# B&R Automation Studio project DeltaTestowa1
Automation Studio 4.12.6.106; technology packages: mapp 5.24.2, mappMotion 5.26.1, mappView 5.24.2

## Configuration Config1

CPU 5APC3100.KBU0-000, AutomationRuntime J4.93, Build 4.1.2, Safety 0.0, Vc V4.73.2

CPU 5APC3100.KBU1-000, AutomationRuntime J4.93, Build 4.1.2, Safety 0.0, Vc V4.73.2

CPU 5APC3100.KBU2-000, AutomationRuntime C4.90, Build 4.1.2, Safety 0.0, Vc 

CPU X20CP1584, AutomationRuntime J4.93, Build 4.1.2, Vc V4.73.2

### Task classes (Cpu.sw)
```
Cyclic#4:
  Program <- Program.prg
Libraries: McBase, MpBase, MpRobotics, McAxGroup, McPathGen, McAxis, McProgInt, McAcpAx, McPureVAx
```

### Task classes (Cpu.sw)
```
Cyclic#1:
  PrgPick <- PickAndPlace.PrgPick.prg
  PrgPickCor <- PickAndPlace.PrgPickCore.prg
  PrgMechs <- PickAndPlace.PrgMechs.prg
  PrgPlace <- PickAndPlace.PrgPlace.prg
Cyclic#4:
  Program <- Program.prg
DataObjects: McAcpSys
NcDataObjects: McDriveLog
Binaries: McAcpDrv, udbdef, McAcpSim, mvLoader, arflatprv, TCData, McProfGen, mCoWebSc, McMechSys, FWRules, arcoal, arsvcreg, Settings, iomap, Config_3, Config_4, Role, ashwac, Config_10, asfw, Config_5, sysconf, Config_2, arconfig, Config_6, Config_8, Config_1, Hierarchy, ashwd, Config_7, User, Config_9
Libraries: UserLib, McBase, MpBase, MpRobotics, McAxGroup, McPathGen, McAxis, McProgInt, McAcpAx, CoTrace, AsZip, FileIO, runtime, MpAxis, asarprof, asieccon, asarlog, asio, asmem, astime, asepl, dataobj, brsystem, arssl, sys_lib, powerlnk, mctrkpath, mppick, MpAlarm
```

### Task classes (Cpu.sw)
```
Cyclic#1:
  PrgPickCor <- PickAndPlace.PrgPickCore.prg
Cyclic#2:
  PrgPick <- PickAndPlace.PrgPick.prg
  PrgPlace <- PickAndPlace.PrgPlace.prg
Cyclic#3:
  PrgMechs <- PickAndPlace.PrgMechs.prg
DataObjects: McAcpSys
NcDataObjects: McDriveLog
Binaries: McAcpDrv, udbdef, McAcpSim, mvLoader, arflatprv, TCData, McProfGen, mCoWebSc, McMechSys, FWRules, arcoal, arsvcreg, OpcUaSrv, Settings, iomap, Config_3, Config_4, Role, ashwac, Config_10, asfw, Config_5, sysconf, Config_2, arconfig, Config_6, Config_8, Config_1, Hierarchy, ashwd, Config_7, User, Config_9
Libraries: UserLib, McBase, MpBase, MpRobotics, McAxGroup, McPathGen, McAxis, McProgInt, McAcpAx, CoTrace, AsZip, FileIO, runtime, MpAxis, McAcpPar, McTrkPath, MpPick, McAcpTrak, MpCnc, MpTool, sys_lib, McDS402Ax, McPureVAx, McStpAx, MpServer, AsIODiag, asarprof, asarlog, asio, asmem, astime, asepl, dataobj, brsystem, arssl, powerlnk, asioacc, aruser, asieccon
```

### Task classes (Cpu1.sw)
```

```

### Task classes (Cpu.sw)
```
Cyclic#4:
  Program <- Program.prg
Libraries: McBase, MpBase, MpRobotics, McAxGroup, McPathGen, McAxis, McProgInt, McAcpAx
```

### Hardware
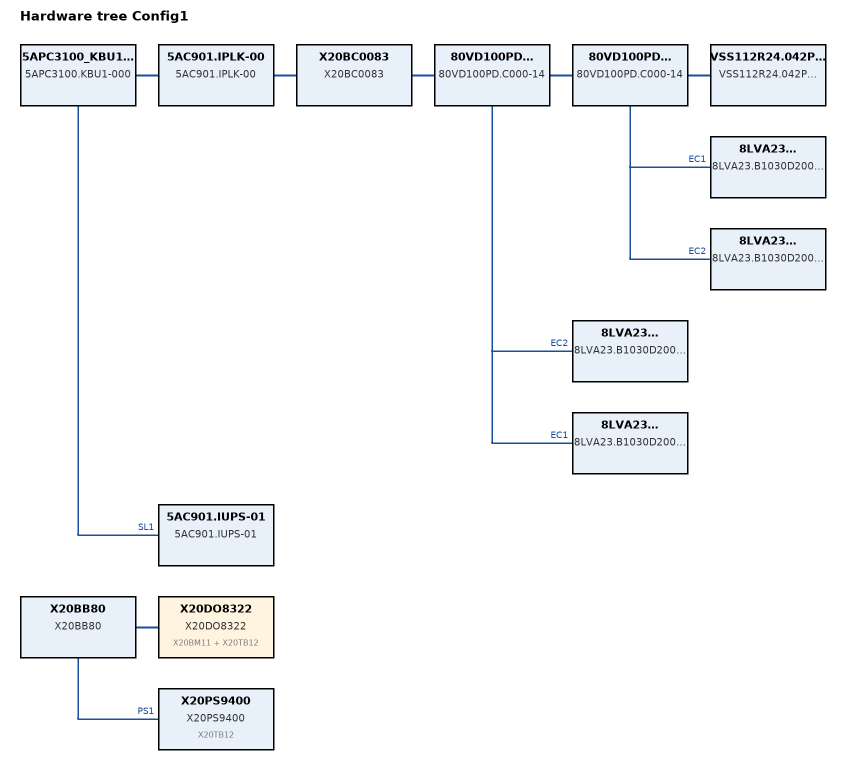
```
5AC901.IPLK-00 : 5AC901.IPLK-00 v1.8.0.1  [SL -> 5APC3100_KBU1_000a.SL2]
  Connector IF1:
    MtuSize = 1500
    CycleTime = 400
    Channel1
    ChannelID1 = McAcpBroadcast
    ChannelType1 = OCTET[36]
    InternetAddress = 192.168.200.240
    SubnetMask = 255.255.255.0
5AC901.IUPS-01 : 5AC901.IUPS-01 v1.3.1.0  [SL -> 5APC3100_KBU1_000a.SL1]
5APC3100_KBU1_000a : 5APC3100.KBU1-000 v2.2.1.0
  Connector IF3:
    AssignedOperatingSystem = ARemb
    ActivateDevice = 1
    Mode = Manual
    InternetAddress = 192.168.0.20
    SubnetMask = 255.255.255.0
    ActivateSnmp = 2
  Connector IF4:
    AssignedOperatingSystem = ARemb
    ActivateDevice = 1
    Mode = Manual
    InternetAddress = 10.0.0.20
    SubnetMask = 255.255.255.0
    ActivateSnmp = 2
  Connector IF5:
    AssignedOperatingSystem = ARemb
  Connector IF6:
    AssignedOperatingSystem = ARemb
  Connector IF7:
    AssignedOperatingSystem = ARemb
  Connector IF8:
    AssignedOperatingSystem = ARemb
  ConfigurationID = Proj_Config1
  MotionLoggerSize = 2048000
  TimerDeviceType = EPLX2X
  TimerDevice = 5AC901.IPLK-00.IF1
  TaskClassIdleTime = 2000
  Cyclic1Tolerance = 0
  FileDevice1
  FileDeviceName1 = CNC_PrgDir
  FileDevicePath1 = C:\CNC_PrgDir\
  FileDevice2
  FileDeviceName2 = CF
  FileDevicePath2 = C:\CF\
  FileDevice3
  FileDeviceName3 = CNC_PrgDirRobot
  FileDevicePath3 = F:\CNC_PrgDirRobot
  ActivateOpcUa = 1
  OpcUaPort = 4841
  OpcUaInformationModels_PV_Version = 1
80VD100PD.C000-14 : 80VD100PD.C000-14 v2.5.0.0  [PLK1 -> 80VD100PD.C000-14a.PLK2 (NodeNumber=1) [Cable Type=PowerlinkCable, Length=10, Version=1.0.0.3]; PLK2 -> VSS112R24.042P-000.PLK1 (NodeNumber=1) [Cable Type=PowerlinkCable, Length=10, Version=1.0.0.3]; EC1 -> 8LVA23.B1030D200-0b.EC; EC2 -> 8LVA23.B1030D200-0c.EC; MT2 -> 8LVA23.B1030D200-0c.MT]
  DriveConfiguration/Module:
    McAcoposTypeID = AcoposMicroDConfig
    ActivateACOPOSSimulationOnPLC = 0
  DriveConfiguration/Channel[1]/RealAxis:
    AxisReference = gAxisQ1
    MechanicalElementsIsInvisible = 0
  DriveConfiguration/Channel[1]/RealAxis/MechanicalElements/Gearbox:
    InputIsReadOnly = 0
    Input = 25
    OutputIsReadOnly = 0
    Output = 1
  DriveConfiguration/Channel[1]/RealAxis/MechanicalElements/RotaryToLinearTransformation:
    ReferenceDistanceIsReadOnly = 0
    ReferenceDistance = 360
  DriveConfiguration/Channel[1]/RealAxis/Controller:
    ModeIsReadOnly = 0
    Mode = PositionController
  DriveConfiguration/Channel[1]/RealAxis/Controller/Mode/Position:
    ProportionalGain = 396.000000
    IntegrationTime = 0.0
    PredictionTime = 0.0004
    TotalDelayTime = 0.0004
  DriveConfiguration/Channel[1]/RealAxis/Controller/Mode/Speed:
    ProportionalGainIsReadOnly = 0
    ProportionalGain = 1.700000
    IntegrationTimeIsReadOnly = 0
    IntegrationTime = 0.0
    FilterTimeIsReadOnly = 0
    FilterTime = 0.0
  DriveConfiguration/Channel[1]/RealAxis/Controller/Mode/LoopFilters:
    LoopFilterXIsReadOnly = 0
    LoopFilter1 = NotUsed
    LoopFilter2 = NotUsed
    LoopFilter3 = NotUsed
  DriveConfiguration/Channel[1]/RealAxis/Homing:
    ModeIsReadOnly = 0
    Mode = Absolute
  DriveConfiguration/Channel[1]/RealAxis/Homing/Mode:
    Position = -472771
  DriveConfiguration/Channel[1]/RealAxis/Homing:
    RestorePositionVariable = 
  DriveConfiguration/Channel[1]/RealAxis/StopReaction:
    QuickstopIsReadOnly = 0
    Quickstop = DecelerationLimit
    DriveErrorIsReadOnly = 0
    DriveError = DecelerationLimit
  DriveConfiguration/Channel[1]/RealAxis/MovementErrorLimits:
    PositionError = 1.0
    VelocityErrorMonitoring = Automatic1
  DriveConfiguration/Channel[1]/RealAxis:
    JerkFilterIsReadOnly = 0
    JerkFilter = NotUsed
    ZeroVibrationFilter = NotUsed
  DriveConfiguration/Channel[1]/RealAxis/DigitalInputs/HomingSwitch:
    SourceIsReadOnly = 0
    Source = NotUsed
    Level = High
  DriveConfiguration/Channel[1]/RealAxis/DigitalInputs/PositiveLimitSwitch:
    SourceIsReadOnly = 0
    Source = NotUsed
    Level = High
  DriveConfiguration/Channel[1]/RealAxis/DigitalInputs/NegativeLimitSwitch:
    SourceIsReadOnly = 0
    Source = NotUsed
    Level = High
  DriveConfiguration/Channel[1]/RealAxis/DigitalInputs/Trigger1:
    Source = X2Trigger1
    Level = High
  DriveConfiguration/Channel[1]/RealAxis/DigitalInputs/Trigger2:
    Source = X2Trigger2
    Level = High
  DriveConfiguration/Channel[1]/RealAxis/DigitalInputs/Quickstop:
    Input = Trigger2
  DriveConfiguration/Channel[1]/RealAxis/Simulation:
    SimulationModeOnPLC = SetValueGeneration
    SimulationModeOnACOPOS = NotUsed
  DriveConfiguration/Channel[2]/RealAxis:
    AxisReference = gAxisQ2
    MechanicalElementsIsInvisible = 0
  DriveConfiguration/Channel[2]/RealAxis/MechanicalElements/Gearbox:
    InputIsReadOnly = 0
    Input = 25
    OutputIsReadOnly = 0
    Output = 1
  DriveConfiguration/Channel[2]/RealAxis/MechanicalElements/RotaryToLinearTransformation:
    ReferenceDistanceIsReadOnly = 0
    ReferenceDistance = 360
  DriveConfiguration/Channel[2]/RealAxis/Controller:
    ModeIsReadOnly = 0
    Mode = PositionController
  DriveConfiguration/Channel[2]/RealAxis/Controller/Mode/Position:
    ProportionalGain = 398.000000
    IntegrationTime = 0.0
    PredictionTime = 0.0004
    TotalDelayTime = 0.0004
  DriveConfiguration/Channel[2]/RealAxis/Controller/Mode/Speed:
    ProportionalGainIsReadOnly = 0
    ProportionalGain = 1.600000
    IntegrationTimeIsReadOnly = 0
    IntegrationTime = 0.0
    FilterTimeIsReadOnly = 0
    FilterTime = 0.0
  DriveConfiguration/Channel[2]/RealAxis/Controller/Mode/LoopFilters:
    LoopFilterXIsReadOnly = 0
    LoopFilter1 = NotUsed
    LoopFilter2 = NotUsed
    LoopFilter3 = NotUsed
  DriveConfiguration/Channel[2]/RealAxis/Homing:
    ModeIsReadOnly = 0
    Mode = Absolute
  DriveConfiguration/Channel[2]/RealAxis/Homing/Mode:
    Position = 77669
  DriveConfiguration/Channel[2]/RealAxis/Homing:
    RestorePositionVariable = 
  DriveConfiguration/Channel[2]/RealAxis/StopReaction:
    QuickstopIsReadOnly = 0
    Quickstop = DecelerationLimit
    DriveErrorIsReadOnly = 0
    DriveError = DecelerationLimit
  DriveConfiguration/Channel[2]/RealAxis/MovementErrorLimits:
    PositionError = 1.0
    VelocityErrorMonitoring = Automatic1
  DriveConfiguration/Channel[2]/RealAxis:
    JerkFilterIsReadOnly = 0
    JerkFilter = NotUsed
    ZeroVibrationFilter = NotUsed
  DriveConfiguration/Channel[2]/RealAxis/DigitalInputs/HomingSwitch:
    SourceIsReadOnly = 0
    Source = NotUsed
    Level = High
  DriveConfiguration/Channel[2]/RealAxis/DigitalInputs/PositiveLimitSwitch:
    SourceIsReadOnly = 0
    Source = NotUsed
    Level = High
  DriveConfiguration/Channel[2]/RealAxis/DigitalInputs/NegativeLimitSwitch:
    SourceIsReadOnly = 0
    Source = NotUsed
    Level = High
  DriveConfiguration/Channel[2]/RealAxis/DigitalInputs/Trigger1:
    Source = X2Trigger1
    Level = High
  DriveConfiguration/Channel[2]/RealAxis/DigitalInputs/Trigger2:
    Source = X2Trigger2
    Level = High
  DriveConfiguration/Channel[2]/RealAxis/DigitalInputs/Quickstop:
    Input = Trigger2
  DriveConfiguration/Channel[2]/RealAxis/Simulation:
    SimulationModeOnPLC = SetValueGeneration
    SimulationModeOnACOPOS = NotUsed
80VD100PD.C000-14a : 80VD100PD.C000-14 v2.5.0.0  [PLK1 -> X20BC0083.PLK2 (NodeNumber=2) [Cable Type=PowerlinkCable, Length=10, Version=1.0.0.3]; PLK2 -> 80VD100PD.C000-14.PLK1 (NodeNumber=2) [Cable Type=PowerlinkCable, Length=10, Version=1.0.0.3]; EC1 -> 8LVA23.B1030D200-0a.EC; EC2 -> 8LVA23.B1030D200-0.EC; MT2 -> 8LVA23.B1030D200-0.MT]
  DriveConfiguration/Module:
    McAcoposTypeID = AcoposMicroDConfig
    ActivateACOPOSSimulationOnPLC = 0
  DriveConfiguration/Channel[1]/RealAxis:
    AxisReference = gAxisQ3
    MechanicalElementsIsInvisible = 0
  DriveConfiguration/Channel[1]/RealAxis/MechanicalElements/Gearbox:
    InputIsReadOnly = 0
    Input = 25
    OutputIsReadOnly = 0
    Output = 1
  DriveConfiguration/Channel[1]/RealAxis/MechanicalElements/RotaryToLinearTransformation:
    ReferenceDistanceIsReadOnly = 0
    ReferenceDistance = 360
  DriveConfiguration/Channel[1]/RealAxis/Controller:
    ModeIsReadOnly = 0
    Mode = PositionController
  DriveConfiguration/Channel[1]/RealAxis/Controller/Mode/Position:
    ProportionalGain = 399.000000
    IntegrationTime = 0.0
    PredictionTime = 0.0004
    TotalDelayTime = 0.0004
  DriveConfiguration/Channel[1]/RealAxis/Controller/Mode/Speed:
    ProportionalGainIsReadOnly = 0
    ProportionalGain = 1.750000
    IntegrationTimeIsReadOnly = 0
    IntegrationTime = 0.0
    FilterTimeIsReadOnly = 0
    FilterTime = 0.0
  DriveConfiguration/Channel[1]/RealAxis/Controller/Mode/LoopFilters:
    LoopFilterXIsReadOnly = 0
    LoopFilter1 = NotUsed
    LoopFilter2 = NotUsed
    LoopFilter3 = NotUsed
  DriveConfiguration/Channel[1]/RealAxis/Homing:
    ModeIsReadOnly = 0
    Mode = Absolute
  DriveConfiguration/Channel[1]/RealAxis/Homing/Mode:
    Position = 3718
  DriveConfiguration/Channel[1]/RealAxis/Homing:
    RestorePositionVariable = 
  DriveConfiguration/Channel[1]/RealAxis/StopReaction:
    QuickstopIsReadOnly = 0
    Quickstop = DecelerationLimit
    DriveErrorIsReadOnly = 0
    DriveError = DecelerationLimit
  DriveConfiguration/Channel[1]/RealAxis/MovementErrorLimits:
    PositionError = 1.0
    VelocityErrorMonitoring = Automatic1
  DriveConfiguration/Channel[1]/RealAxis:
    JerkFilterIsReadOnly = 0
    JerkFilter = NotUsed
    ZeroVibrationFilter = NotUsed
  DriveConfiguration/Channel[1]/RealAxis/DigitalInputs/HomingSwitch:
    SourceIsReadOnly = 0
    Source = NotUsed
    Level = High
  DriveConfiguration/Channel[1]/RealAxis/DigitalInputs/PositiveLimitSwitch:
    SourceIsReadOnly = 0
    Source = NotUsed
    Level = High
  DriveConfiguration/Channel[1]/RealAxis/DigitalInputs/NegativeLimitSwitch:
    SourceIsReadOnly = 0
    Source = NotUsed
    Level = High
  DriveConfiguration/Channel[1]/RealAxis/DigitalInputs/Trigger1:
    Source = X2Trigger1
    Level = High
  DriveConfiguration/Channel[1]/RealAxis/DigitalInputs/Trigger2:
    Source = X2Trigger2
    Level = High
  DriveConfiguration/Channel[1]/RealAxis/DigitalInputs/Quickstop:
    Input = Trigger2
  DriveConfiguration/Channel[1]/RealAxis/Simulation:
    SimulationModeOnPLC = SetValueGeneration
    SimulationModeOnACOPOS = NotUsed
  DriveConfiguration/Channel[2]/RealAxis:
    AxisReference = gAxis_1
    MechanicalElementsIsInvisible = 0
  DriveConfiguration/Channel[2]/RealAxis/MechanicalElements/Gearbox:
    InputIsReadOnly = 0
    Input = 2
    OutputIsReadOnly = 0
    Output = 1
  DriveConfiguration/Channel[2]/RealAxis/MechanicalElements/RotaryToLinearTransformation:
    ReferenceDistanceIsReadOnly = 0
    ReferenceDistance = 136
  DriveConfiguration/Channel[2]/RealAxis/Controller:
    ModeIsReadOnly = 0
    Mode = PositionController
  DriveConfiguration/Channel[2]/RealAxis/Controller/Mode/Position:
    ProportionalGain = 374.000000
    IntegrationTime = 0.0
    PredictionTime = 0.0004
    TotalDelayTime = 0.0004
  DriveConfiguration/Channel[2]/RealAxis/Controller/Mode/Speed:
    ProportionalGainIsReadOnly = 0
    ProportionalGain = 0.950000
    IntegrationTimeIsReadOnly = 0
    IntegrationTime = 0.0
    FilterTimeIsReadOnly = 0
    FilterTime = 0.0
  DriveConfiguration/Channel[2]/RealAxis/Controller/Mode/LoopFilters:
    LoopFilterXIsReadOnly = 0
    LoopFilter1 = NotUsed
    LoopFilter2 = NotUsed
    LoopFilter3 = NotUsed
  DriveConfiguration/Channel[2]/RealAxis/Homing:
    ModeIsReadOnly = 0
    Mode = Direct
  DriveConfiguration/Channel[2]/RealAxis/Homing/Mode:
    Position = 0.0
    ReferencePulse = NotUsed
  DriveConfiguration/Channel[2]/RealAxis/Homing:
    RestorePositionVariable = 
  DriveConfiguration/Channel[2]/RealAxis/StopReaction:
    QuickstopIsReadOnly = 0
    Quickstop = DecelerationLimit
    DriveErrorIsReadOnly = 0
    DriveError = DecelerationLimit
  DriveConfiguration/Channel[2]/RealAxis/MovementErrorLimits:
    PositionError = 1.0
    VelocityErrorMonitoring = Automatic1
  DriveConfiguration/Channel[2]/RealAxis:
    JerkFilterIsReadOnly = 0
    JerkFilter = NotUsed
    ZeroVibrationFilter = NotUsed
  DriveConfiguration/Channel[2]/RealAxis/DigitalInputs/HomingSwitch:
    SourceIsReadOnly = 0
    Source = NotUsed
    Level = High
  DriveConfiguration/Channel[2]/RealAxis/DigitalInputs/PositiveLimitSwitch:
    SourceIsReadOnly = 0
    Source = NotUsed
    Level = High
  DriveConfiguration/Channel[2]/RealAxis/DigitalInputs/NegativeLimitSwitch:
    SourceIsReadOnly = 0
    Source = NotUsed
    Level = High
  DriveConfiguration/Channel[2]/RealAxis/DigitalInputs/Trigger1:
    Source = X2Trigger1
    Level = High
  DriveConfiguration/Channel[2]/RealAxis/DigitalInputs/Trigger2:
    Source = X2Trigger2
    Level = High
  DriveConfiguration/Channel[2]/RealAxis/DigitalInputs/Quickstop:
    Input = Trigger2
  DriveConfiguration/Channel[2]/RealAxis/Simulation:
    SimulationModeOnPLC = SetValueGeneration
    SimulationModeOnACOPOS = NotUsed
8LVA23.B1030D200-0 : 8LVA23.B1030D200-0 v2.2.0.3  [EC -> 80VD100PD.C000-14a.EC2; MT -> 80VD100PD.C000-14a.MT2]
  M1/MotorParameters:
    MOTOR_AMB_TEMP_RATED = 40
8LVA23.B1030D200-0a : 8LVA23.B1030D200-0 v2.2.0.3  [EC -> 80VD100PD.C000-14a.EC1; MT -> 80VD100PD.C000-14a.MT1]
  M1/MotorParameters:
    MOTOR_AMB_TEMP_RATED = 40
8LVA23.B1030D200-0b : 8LVA23.B1030D200-0 v2.2.0.3  [EC -> 80VD100PD.C000-14.EC1; MT -> 80VD100PD.C000-14.MT1]
  M1/MotorParameters:
    MOTOR_AMB_TEMP_RATED = 40
8LVA23.B1030D200-0c : 8LVA23.B1030D200-0 v2.2.0.3  [EC -> 80VD100PD.C000-14.EC2; MT -> 80VD100PD.C000-14.MT2]
  M1/MotorParameters:
    MOTOR_AMB_TEMP_RATED = 40
VSS112R24.042P-000 : VSS112R24.042P-000 v1.9.0.730  [PLK1 -> 80VD100PD.C000-14.PLK2 (NodeNumber=4) [Cable Type=PowerlinkCable, Length=10, Version=1.0.0.3]]
  VisionConfig = gCamera
X20BB80 : X20BB80 v1.1.0.0
X20BC0083 : X20BC0083 v2.14.0.0  [PLK1 -> 5AC901.IPLK-00.IF1 (NodeNumber=3) [Cable Type=PowerlinkCable, Length=10, Version=1.0.0.3]; PLK2 -> 80VD100PD.C000-14a.PLK1 (NodeNumber=3) [Cable Type=PowerlinkCable, Length=10, Version=1.0.0.3]; SL -> X20BB80.SL1]
X20BM11 : X20BM11 v1.1.0.0  [X2X1 -> X20BB80.IF1]
X20DO8322 : X20DO8322 v1.5.0.0  [SS1 -> X20TB12a.SS; SL -> X20BM11.SL1]
X20PS9400 : X20PS9400 v1.8.0.0  [SS1 -> X20TB12.SS; PS -> X20BB80.PS1]
X20TB12 : X20TB12 v1.0.0.0
X20TB12a : X20TB12 v1.0.0.0
```

### Config_4.axesgroupfeature - 5APC3100_KBU0_000/mappMotion/4AxesDeltaA/Config_4.axesgroupfeature
```
Element Feature_Programs (Type=axesgroupfeature)
  Type = Program
    ModalDataBehaviour = UseAxesGroupSettings
    InitialSettings:
      InterpolationTypes = LinearRapid
      PositionCoordinates = Absolute
      CircleCoordinates = Relative
      JACS_ACSProgramming = JACS
      ContourConnection = Inactive
      ProgrammingUnits = UseAxesGroupSettings
      Feedrates:
        FeedPath = Standard
        FeedCharacteristic = StandardCharacteristic
        FeedType = Feedrate
        FeedReduction = Inactive
        FeedrateValue = 0.0
        InverseFeedrateValue = 0.0
        FeedratePerRevValue = 0.0
    DefaultLanguage = BRGCode
    Location = Default
      FileDevice = CNC_PrgDir
Element Feature_Jogging (Type=axesgroupfeature)
  Type = Jogging
Element Feature_Tracking (Type=axesgroupfeature)
  Type = Tracking
    ModalDataBehaviour = UseAxesGroupSettings
    SynchronisationGeometry = Basic
      CartesianRadius = 20
    TorqueLimitConsideration = Exact
Element Feature_FrameHierarchy (Type=axesgroupfeature)
  Type = FrameHierarchy
    ModalDataBehaviour = UseAxesGroupSettings
    FrameHierarchy = Custom
      FramePropertyMapping:
        BCS = RoboBase
        PCS = ZeroPosPickConveyor
        SCS1
        SCS2
        SCS3
        SCS4
        SCS5
      MCS:
        Name = MachineBase
        Frame[1]:
          Name = RoboBase
          Type = StandardFrame
            Translation:
              X = 0.0
              Y = 0.0
              Z = 150
            Orientation:
              Angle1 = 0.0
              Angle2 = 0.0
              Angle3 = 0.0
          Frame[1]:
            Name = ZeroPosPickConveyor
            Type = StandardFrame
              Translation:
                X = 0.0
                Y = 400
                Z = -1000
              Orientation:
                Angle1 = 0.0
                Angle2 = 0.0
                Angle3 = 0.0
Element Feature_PatchDefinition (Type=axesgroupfeature)
  Type = PathDefinitions
    ModalDataBehaviour = UseAxesGroupSettings
    PathDefinition[1]:
      Name = Path1
      Type = CartesianPath
        CalculatedIn = PCS
      Limit = Internal
        Velocity = NotUsed
        Acceleration = NotUsed
        Deceleration = NotUsed
        Jerk = NotUsed
```

### Config_10.purevaxcfg - 5APC3100_KBU0_000/mappMotion/Config_10.purevaxcfg
```
Element PureVAxCfg_1 (Type=purevaxcfg)
  TypeID = PureVAxConfig
  PureVAxis:
    AxisReference
    Homing:
      Mode = Direct
        Position = 0.0
        ReferencePulse = NotUsed
      RestorePositionVariable
    JerkFilter = NotUsed
    ZeroVibrationFilter = NotUsed
```

### Config_11.purevaxcfg - 5APC3100_KBU0_000/mappMotion/Config_11.purevaxcfg
```
Element PureVAxCfg_2 (Type=purevaxcfg)
  TypeID = PureVAxConfig
  PureVAxis:
    AxisReference
    Homing:
      Mode = Direct
        Position = 0.0
        ReferencePulse = NotUsed
      RestorePositionVariable
    JerkFilter = NotUsed
    ZeroVibrationFilter = NotUsed
```

### IoMap.iom - 5APC3100_KBU1_000a/IoMap.iom
```iecst
VAR_CONFIG
	::PrgPickCor:Gripper AT %QX."X20DO8322".DigitalOutput08;
	::Vision:Cam.Parameters.SetFocus AT %QW."VSS112R24.042P-000".SetFocus;
	::Vision:Cam.Parameters.ExposureTime AT %QD."VSS112R24.042P-000".ExposureTime01;
	::Vision:Cam.Parameters.FlashColor AT %QB."VSS112R24.042P-000".FlashColor01;
	::Vision:Cam.Parameters.FlashSegment AT %QB."VSS112R24.042P-000".FlashSegment01;
	::Vision:Cam.Camera_Output.PosMatchX AT %ID."VSS112R24.042P-000".PositionXMatching01;
	::Vision:Cam.Camera_Output.PosMatchY AT %ID."VSS112R24.042P-000".PositionYMatching01;
	::Vision:Cam.Cmd.Enable_Matching AT %QX."VSS112R24.042P-000".EnableMatching;
	::Vision:CameraStatus AT %ID."VSS112R24.042P-000".CameraStatus;
	::Vision:Cam.Status.IsCameraReady AT %IX."VSS112R24.042P-000".ImageAcquisitionReady;
	::Vision:Cam.Camera_Output.NumResults AT %IB."VSS112R24.042P-000".NumResultsMatching;
	::Vision:Cam.Camera_Output.PhotosNum AT %IB."VSS112R24.042P-000".CompletedAcquisitionCnt;
	::Vision:Cam.Camera_Output.ProcesingTime AT %IW."VSS112R24.042P-000".CameraProcessingTime;
	::gIsCameraActive AT %IX."VSS112R24.042P-000".ImageProcessingActive;
END_VAR
```

### Config_1.axesgroup - 5APC3100_KBU1_000a/mappMotion/4AxesDeltaA/Config_1.axesgroup
```
Element g4AxDeltaA (Type=axesgroup)
  Type = PathGenAxesGroup
    ProcessingTaskClass = 255
    License = 1
    PhysicalAxes:
      JointAxes:
        JointAxisAxisRefIsReadOnly = 0
        JointAxis[1]:
          Name = Q1
          AxisRef = gAxisQ1
        JointAxis[2]:
          Name = Q2
          AxisRef = gAxisQ2
        JointAxis[3]:
          Name = Q3
          AxisRef = gAxisQ3
        JointAxis[4]:
          Name = Q4
          AxisRef = gAxisQ4
    MechanicalSystem:
      MechSysRefIsReadOnly = 0
      MechSysRef = MechSys_4AxDeltaA
    BasicSettings:
      ModalDataBehaviour = ResetToDefault
      GeometryPlanning:
        TCPResolutionIsReadOnly = 0
        TCPResolution:
          LengthResolution = 0.001
          AngleResolution = 0.001
        Rounding:
          PathDistance = 0.0
          SymmetricRounding = Yes
          LastSegment = Half
          AvoidZeroCurvature = No
        RoundingMode = Standard
        MaxCornerDeviation = 0.0
        MaxTangentialTransitionDeviation = 0.0
        MaxRadiusDeviation = 0.001
        WorkingPlane = XY
      TrajectoryPlanningIsReadOnly = 0
      TrajectoryPlanning = Basic
        LimitCheckResolutionIsReadOnly = 0
        LimitCheckResolution = Automatic
        BufferTime = Automatic
        BarrierParametrization = JointCoordinates
      Miscellaneous:
        NonMovementsLimit = NotUsed
        TimeStretchOverride:
          JerkSuppression = NotUsed
    AxesGroupFeatures:
      FeatureRef[1] = Feature_FrameHierarchy
      FeatureRef[2] = Feature_Jogging
      FeatureRef[3] = Feature_PathDefinition
      FeatureRef[4] = Feature_Programs
      FeatureRef[5] = Feature_Tracking
      FeatureRef[6] = Feature_MotionPacketLog
  Alarms = MpAlarmX
```

### Config_2.axis - 5APC3100_KBU1_000a/mappMotion/4AxesDeltaA/Config_2.axis
```
Element gAxisQ1 (Type=axis)
  BaseTypeIsReadOnly = 0
  BaseType = RotaryBounded
    MeasurementUnitIsReadOnly = 0
    MeasurementUnit = 17476
    MeasurementResolutionIsReadOnly = 0
    MeasurementResolution = 0.01
    CountDirectionIsReadOnly = 0
    CountDirection = Standard
  MovementLimitsIsReadOnly = 0
  MovementLimits = Internal
    Position:
      LowerLimitMin = -1.79769313486231E308
      UpperLimitMax = 1.79769313486231E308
      LowerLimit = -30
      UpperLimit = 110
    VelocityIsReadOnly = 0
    Velocity:
      VelocityMax = 3.4E38
      Velocity = 50000
    AccelerationIsReadOnly = 0
    Acceleration:
      AccelerationMax = 3.4E38
      Acceleration = 500000
    DecelerationIsReadOnly = 0
    Deceleration:
      DecelerationMax = 3.4E38
      Deceleration = 500000
  Alarms = MpAlarmX
    mapp.AlarmX.Core.Configuration:
      [0]:
        Message = System problem - axis Q1
      [1]:
        Message = Initialization problem - axis Q1
      [2]:
        Message = Parameter problem - axis Q1
      [3]:
        Message = Operation problem - axis Q1
      [4]:
        Message = Data access problem - axis Q1
      [5]:
        Message = Syntax error - axis Q1
      [9]:
        Message = Network problem - axis Q1
      [10]:
        Message = Encoder problem - axis Q1
      [11]:
        Message = Drive problem - axis Q1
      [12]:
        Message = IO problem - axis Q1
      [13]:
        Message = Supply problem - axis Q1
      [14]:
        Message = Motor problem - axis Q1
      [15]:
        Message = Holding brake problem - axis Q1
      [19]:
        Message = Movement error limit reached - axis Q1
      [20]:
        Message = HW or SW movement limits reached - axis Q1
      [21]:
        Message = Enable input low - axis Q1
Element gAxisQ2 (Type=axis)
  BaseTypeIsReadOnly = 0
  BaseType = RotaryBounded
    MeasurementUnitIsReadOnly = 0
    MeasurementUnit = 17476
    MeasurementResolutionIsReadOnly = 0
    MeasurementResolution = 0.01
    CountDirectionIsReadOnly = 0
    CountDirection = Inverse
  MovementLimitsIsReadOnly = 0
  MovementLimits = Internal
    Position:
      LowerLimitMin = -1.79769313486231E308
      UpperLimitMax = 1.79769313486231E308
      LowerLimit = -30
      UpperLimit = 110
    VelocityIsReadOnly = 0
    Velocity:
      VelocityMax = 3.4E38
      Velocity = 50000
    AccelerationIsReadOnly = 0
    Acceleration:
      AccelerationMax = 3.4E38
      Acceleration = 500000
    DecelerationIsReadOnly = 0
    Deceleration:
      DecelerationMax = 3.4E38
      Deceleration = 500000
  Alarms = MpAlarmX
    mapp.AlarmX.Core.Configuration:
      [0]:
        Message = System problem - axis Q2
      [1]:
        Message = Initialization problem - axis Q2
      [2]:
        Message = Parameter problem - axis Q2
      [3]:
        Message = Operation problem - axis Q2
      [4]:
        Message = Data access problem - axis Q2
      [5]:
        Message = Syntax error - axis Q2
      [9]:
        Message = Network problem - axis Q2
      [10]:
        Message = Encoder problem - axis Q2
      [11]:
        Message = Drive problem - axis Q2
      [12]:
        Message = IO problem - axis Q2
      [13]:
        Message = Supply problem - axis Q2
      [14]:
        Message = Motor problem - axis Q2
      [15]:
        Message = Holding brake problem - axis Q2
      [19]:
        Message = Movement error limit reached - axis Q2
      [20]:
        Message = HW or SW movement limits reached - axis Q2
      [21]:
        Message = Enable input low - axis Q2
Element gAxisQ3 (Type=axis)
  BaseTypeIsReadOnly = 0
  BaseType = RotaryBounded
    MeasurementUnitIsReadOnly = 0
    MeasurementUnit = 17476
    MeasurementResolutionIsReadOnly = 0
    MeasurementResolution = 0.01
    CountDirectionIsReadOnly = 0
    CountDirection = Inverse
  MovementLimitsIsReadOnly = 0
  MovementLimits = Internal
    Position:
      LowerLimitMin = -1.79769313486231E308
      UpperLimitMax = 1.79769313486231E308
      LowerLimit = -30
      UpperLimit = 110
    VelocityIsReadOnly = 0
    Velocity:
      VelocityMax = 3.4E38
      Velocity = 50000
    AccelerationIsReadOnly = 0
    Acceleration:
      AccelerationMax = 3.4E38
      Acceleration = 500000
    DecelerationIsReadOnly = 0
    Deceleration:
      DecelerationMax = 3.4E38
      Deceleration = 500000
  Alarms = MpAlarmX
    mapp.AlarmX.Core.Configuration:
      [0]:
        Message = System problem - axis Q3
      [1]:
        Message = Initialization problem - axis Q3
      [2]:
        Message = Parameter problem - axis Q3
      [3]:
        Message = Operation problem - axis Q3
      [4]:
        Message = Data access problem - axis Q3
      [5]:
        Message = Syntax error - axis Q3
      [9]:
        Message = Network problem - axis Q3
      [10]:
        Message = Encoder problem - axis Q3
      [11]:
        Message = Drive problem - axis Q3
      [12]:
        Message = IO problem - axis Q3
      [13]:
        Message = Supply problem - axis Q3
      [14]:
        Message = Motor problem - axis Q3
      [15]:
        Message = Holding brake problem - axis Q3
      [19]:
        Message = Movement error limit reached - axis Q3
      [20]:
        Message = HW or SW movement limits reached - axis Q3
      [21]:
        Message = Enable input low - axis Q3
Element gAxisQ4 (Type=axis)
  BaseTypeIsReadOnly = 0
  BaseType = Rotary
    MeasurementUnitIsReadOnly = 0
    MeasurementUnit = 17476
    MeasurementResolutionIsReadOnly = 0
    MeasurementResolution = 0.01
    CountDirectionIsReadOnly = 0
    CountDirection = Standard
  MovementLimitsIsReadOnly = 0
  MovementLimits = InternalForPathControlledAxis
    Position:
      LowerLimitMin = -1.79769313486231E308
      UpperLimitMax = 1.79769313486231E308
      LowerLimit = -1000.0
      UpperLimit = 1000.0
    VelocityIsReadOnly = 0
    Velocity:
      VelocityMax = 3.4E38
      Velocity = 50000
    AccelerationIsReadOnly = 0
    Acceleration:
      AccelerationMax = 3.4E38
      Acceleration = 500000
    DecelerationIsReadOnly = 0
    Deceleration:
      DecelerationMax = 3.4E38
      Deceleration = 500000
    JerkIsReadOnly = 0
    TorqueIsInvisible = 0
    TorqueIsReadOnly = 0
  Alarms = MpAlarmX
    mapp.AlarmX.Core.Configuration:
      [0]:
        Message = System problem - axis Q4
      [1]:
        Message = Initialization problem - axis Q4
      [2]:
        Message = Parameter problem - axis Q4
      [3]:
        Message = Operation problem - axis Q4
      [4]:
        Message = Data access problem - axis Q4
      [5]:
        Message = Syntax error - axis Q4
      [9]:
        Message = Network problem - axis Q4
      [10]:
        Message = Encoder problem - axis Q4
      [11]:
        Message = Drive problem - axis Q4
      [12]:
        Message = IO problem - axis Q4
      [13]:
        Message = Supply problem - axis Q4
      [14]:
        Message = Motor problem - axis Q4
      [15]:
        Message = Holding brake problem - axis Q4
      [19]:
        Message = Movement error limit reached - axis Q4
      [20]:
        Message = HW or SW movement limits reached - axis Q4
      [21]:
        Message = Enable input low - axis Q4
```

### Config_3.mechanicalsystem - 5APC3100_KBU1_000a/mappMotion/4AxesDeltaA/Config_3.mechanicalsystem
```
Element MechSys_4AxDeltaA (Type=mechanicalsystem)
  TypeIsReadOnly = 0
  Type = Delta
    SubtypeIsReadOnly = 0
    Subtype = 4AxesDeltaA
      SceneViewerObject = Generic
      DescriptionIsReadOnly = 0
      Description = Standard
        Dimensions:
          BasePlatform:
            CenterIsReadOnly = 0
            Center:
              X = 0.0
              Y = 0.0
              Z = 0.0
            ArmLinkPointIsReadOnly = 0
            Arm1LinkPoint:
              Angle = -90
              Radius = 150
              Z = 0.0
            Arm2LinkPoint:
              Angle = 0
              Radius = 138
              Z = 80
            Arm3LinkPoint:
              Angle = 90
              Radius = 150
              Z = 0
          Arms:
            ArmIsReadOnly = 0
            Arm1:
              UpperArmLength = 150
              LowerArmLength = 435
            Arm2:
              UpperArmLength = 150
              LowerArmLength = 435
            Arm3:
              UpperArmLength = 150
              LowerArmLength = 435
            LowerArmPairDistance = 90
          EndEffectorPlatform:
            ArmLinkPointIsReadOnly = 0
            Arm1LinkPoint:
              Radius = 80
              Z = 0.0
            Arm2LinkPoint:
              Radius = 70
              Z = 0
            Arm3LinkPoint:
              Radius = 80
              Z = 0.0
            TranslationToFlangeIsReadOnly = 0
            TranslationToFlange:
              X = 0.0
              Y = 0.0
              Z = -45
        Offsets:
          JointAxisIsReadOnly = 0
          JointAxis[1] = -20
          JointAxis[2] = 0.0
          JointAxis[3] = -20
          JointAxis[4] = 0.0
        CountDirections:
          JointAxisIsReadOnly = 0
          JointAxis[1] = Standard
          JointAxis[2] = Standard
          JointAxis[3] = Standard
          JointAxis[4] = Standard
      CoordinatesNames = Default
        XCoordinateName = X
        YCoordinateName = Y
        ZCoordinateName = Z
        CCoordinateName = C
      TcpOrientation:
        Frames = Used
      WireFrameModelIsReadOnly = 0
      WireFrameModel = Standard
        UpperArm1IsReadOnly = 0
        UpperArm1 = ConnectionLine
          DistanceMin = -1.79769313486231E308
          DistanceMax = 1.79769313486231E308
          Distance = 0.0
        LowerArm1IsReadOnly = 0
        LowerArm1 = ConnectionLine
          DistanceMin = -1.79769313486231E308
          DistanceMax = 1.79769313486231E308
          Distance = 0.0
        UpperArm2IsReadOnly = 0
        UpperArm2 = ConnectionLine
          DistanceMin = -1.79769313486231E308
          DistanceMax = 1.79769313486231E308
          Distance = 0.0
        LowerArm2IsReadOnly = 0
        LowerArm2 = ConnectionLine
          DistanceMin = -1.79769313486231E308
          DistanceMax = 1.79769313486231E308
          Distance = 0.0
        UpperArm3IsReadOnly = 0
        UpperArm3 = ConnectionLine
          DistanceMin = -1.79769313486231E308
          DistanceMax = 1.79769313486231E308
          Distance = 0.0
        LowerArm3IsReadOnly = 0
        LowerArm3 = ConnectionLine
          DistanceMin = -1.79769313486231E308
          DistanceMax = 1.79769313486231E308
          Distance = 0.0
        EndEffectorPlatformToFlangeIsReadOnly = 0
        EndEffectorPlatformToFlange = ConnectionLine
          DistanceMin = -1.79769313486231E308
          DistanceMax = 1.79769313486231E308
          Distance = 1
        FlangeToTcp = ConnectionLine
          DistanceMin = -1.79769313486231E308
          DistanceMax = 1.79769313486231E308
          Distance = 45
      DynamicModelIsReadOnly = 0
      DynamicModel = DynParTable
        TableRef
      InternalDynamicModelIsReadOnly = 0
      InternalDynamicModel = NotUsed
      DynamicLimits = DynParTables
        GearboxLimitsTableRef
        CrossSectionLimitsTableRef
      InternalDynamicLimits = NotUsed
      LoadDependentJerkLimitsIsReadOnly = 0
      LoadDependentJerkLimits = NotUsed
      CouplingsIsInvisible = 0
      JointAxesPositionLimits:
        JointAxisIsReadOnly = 0
        JointAxis[1] = UseAxisLimits
        JointAxis[2] = UseAxisLimits
        JointAxis[3] = UseAxisLimits
        JointAxis[4] = UseAxisLimits
      WorkingRangeIsReadOnly = 0
      WorkingRange = NotUsed
```

### Config_4.axesgroupfeature - 5APC3100_KBU1_000a/mappMotion/4AxesDeltaA/Config_4.axesgroupfeature
```
Element Feature_Programs (Type=axesgroupfeature)
  Type = Program
    ModalDataBehaviour = UseAxesGroupSettings
    InitialSettings:
      InterpolationTypes = LinearRapid
      PositionCoordinates = Absolute
      CircleCoordinates = Relative
      JACS_ACSProgramming = JACS
      ContourConnection = Inactive
      ProgrammingUnits = UseAxesGroupSettings
      Feedrates:
        FeedPath = Standard
        FeedCharacteristic = StandardCharacteristic
        FeedType = Feedrate
        FeedReduction = Inactive
        FeedrateValue = 0.0
        InverseFeedrateValue = 0.0
        FeedratePerRevValue = 0.0
    DefaultLanguage = BRGCode
    Location = User
      UserLocation[1]:
        FileDevice = CNC_PrgDir
      UserLocation[2]:
        FileDevice = CNC_PrgDirRobot
Element Feature_Jogging (Type=axesgroupfeature)
  Type = Jogging
Element Feature_MotionPacketLog (Type=axesgroupfeature)
  Type = MotionPacketLog
    Location = User
      FileDevice = CNC_PrgDir
```

### Config_10.purevaxcfg - 5APC3100_KBU1_000a/mappMotion/Config_10.purevaxcfg
```
Element PureVAxCfg_1 (Type=purevaxcfg)
  TypeID = PureVAxConfig
  PureVAxis:
    AxisReference = gAxisQ4
    Homing:
      Mode = Direct
        Position = 0.0
        ReferencePulse = NotUsed
      RestorePositionVariable
    JerkFilter = NotUsed
    ZeroVibrationFilter = NotUsed
Element PureVAxCfg_2 (Type=purevaxcfg)
  TypeID = PureVAxConfig
  PureVAxis:
    AxisReference = gAxis_2
    Homing:
      Mode = Direct
        Position = 0.0
        ReferencePulse = NotUsed
      RestorePositionVariable
    JerkFilter = NotUsed
    ZeroVibrationFilter = NotUsed
```

### Config_5.axis - 5APC3100_KBU1_000a/mappMotion/PnP_AddOn/Config_5.axis
```
Element gAxis_1 (Type=axis)
  BaseTypeIsReadOnly = 0
  BaseType = LinearPeriodic
    MeasurementUnit = 5066068
    MeasurementResolutionIsReadOnly = 0
    MeasurementResolution = 0.01
    CountDirectionIsReadOnly = 0
    CountDirection = Inverse
    PeriodSettings:
      Period = 2000
  MovementLimitsIsReadOnly = 0
  MovementLimits = Internal
    Position:
      LowerLimitMin = -1.79769313486231E308
      UpperLimitMax = 1.79769313486231E308
      LowerLimit = -1000.0
      UpperLimit = 1000.0
    VelocityIsReadOnly = 0
    Velocity:
      VelocityMax = 3.4E38
      Velocity = 50
    AccelerationIsReadOnly = 0
    Acceleration:
      AccelerationMax = 3.4E38
      Acceleration = 20
    DecelerationIsReadOnly = 0
    Deceleration:
      DecelerationMax = 3.4E38
      Deceleration = 20
  Alarms = MpAlarmX
    mapp.AlarmX.Core.Configuration:
      [0]:
        Message = System problem - ConveyorPick
      [1]:
        Message = Initialization problem - ConveyorPick
      [2]:
        Message = Parameter problem - ConveyorPick
      [3]:
        Message = Operation problem - ConveyorPick
      [4]:
        Message = Data access problem - ConveyorPick
      [5]:
        Message = Syntax error - ConveyorPick
      [9]:
        Message = Network problem - ConveyorPick
      [10]:
        Message = Encoder problem - ConveyorPick
      [11]:
        Message = Drive problem - ConveyorPick
      [12]:
        Message = IO problem - ConveyorPick
      [13]:
        Message = Supply problem - ConveyorPick
      [14]:
        Message = Motor problem - ConveyorPick
      [15]:
        Message = Holding brake problem - ConveyorPick
      [19]:
        Message = Movement error limit reached - ConveyorPick
      [20]:
        Message = HW or SW movement limits reached - ConveyorPick
      [21]:
        Message = Enable input low - ConveyorPick
Element gAxis_2 (Type=axis)
  BaseTypeIsReadOnly = 0
  BaseType = LinearPeriodic
    MeasurementUnit = 5066068
    MeasurementResolutionIsReadOnly = 0
    MeasurementResolution = 0.01
    CountDirectionIsReadOnly = 0
    CountDirection = Standard
    PeriodSettings:
      Period = 2000
  MovementLimitsIsReadOnly = 0
  MovementLimits = Internal
    Position:
      LowerLimitMin = -1.79769313486231E308
      UpperLimitMax = 1.79769313486231E308
      LowerLimit = -1000.0
      UpperLimit = 1000.0
    VelocityIsReadOnly = 0
    Velocity:
      VelocityMax = 3.4E38
      Velocity = 1
    AccelerationIsReadOnly = 0
    Acceleration:
      AccelerationMax = 3.4E38
      Acceleration = 1
    DecelerationIsReadOnly = 0
    Deceleration:
      DecelerationMax = 3.4E38
      Deceleration = 1
  Alarms = MpAlarmX
    mapp.AlarmX.Core.Configuration:
      [0]:
        Message = System problem - PlaceHolder
      [1]:
        Message = Initialization problem - PlaceHolder
      [2]:
        Message = Parameter problem - PlaceHolder
      [3]:
        Message = Operation problem - PlaceHolder
      [4]:
        Message = Data access problem - PlaceHolder
      [5]:
        Message = Syntax error - PlaceHolder
      [9]:
        Message = Network problem - PlaceHolder
      [10]:
        Message = Encoder problem - PlaceHolder
      [11]:
        Message = Drive problem - PlaceHolder
      [12]:
        Message = IO problem - PlaceHolder
      [13]:
        Message = Supply problem - PlaceHolder
      [14]:
        Message = Motor problem - PlaceHolder
      [15]:
        Message = Holding brake problem - PlaceHolder
      [19]:
        Message = Movement error limit reached - PlaceHolder
      [20]:
        Message = HW or SW movement limits reached - PlaceHolder
      [21]:
        Message = Enable input low - PlaceHolder
```

### Config_6.axesgroupfeature - 5APC3100_KBU1_000a/mappMotion/PnP_AddOn/Config_6.axesgroupfeature
```
Element Feature_FrameHierarchy (Type=axesgroupfeature)
  Type = FrameHierarchy
    ModalDataBehaviour = UseAxesGroupSettings
    FrameHierarchy = Custom
      FramePropertyMapping:
        BCS = RoboBase
        PCS = ZeroPosPickConveyor
        SCS1
        SCS2
        SCS3
        SCS4
        SCS5
      MCS:
        Name = MachineBase
        Frame[1]:
          Name = RoboBase
          Type = StandardFrame
            Translation:
              X = 0.0
              Y = 0
              Z = 490
            Orientation:
              Angle1 = 0.0
              Angle2 = 0.0
              Angle3 = 0.0
          Frame[1]:
            Name = ZeroPosPickConveyor
            Type = StandardFrame
              Translation:
                X = 0.0
                Y = 400
                Z = -1000
              Orientation:
                Angle1 = 0.0
                Angle2 = 0.0
                Angle3 = 0.0
Element Feature_Tracking (Type=axesgroupfeature)
  Type = Tracking
    ModalDataBehaviour = UseAxesGroupSettings
    SynchronisationGeometry = Basic
      CartesianRadius = 20.0
    TorqueLimitConsideration = Exact
Element Feature_PathDefinition (Type=axesgroupfeature)
  Type = PathDefinitions
    ModalDataBehaviour = UseAxesGroupSettings
    PathDefinition[1]:
      Name = Path1
      Type = CartesianPath
        CalculatedIn = PCS
      Limit = Internal
        Velocity = NotUsed
        Acceleration = NotUsed
        Deceleration = NotUsed
        Jerk = NotUsed
```

### Config_7.pickobjectlist - 5APC3100_KBU1_000a/mappMotion/PnP_AddOn/Config_7.pickobjectlist
```
Element gPickObjectList_1 (Type=pickobjectlist)
  Object[1] = SingleItem
    Name = MyProduct
  Object[2] = Container
    Name = MyContainer
    Layer[1]:
      Position[1]:
        Object = MyProduct
        Translation:
          X = 0.0
          Y = 0.0
          Z = 0.0
        Orientation:
          Angle1 = 0.0
          Angle2 = 0.0
          Angle3 = 0.0
      Position[2]:
        Object = MyProduct
        Translation:
          X = 48.0
          Y = 0.0
          Z = 0.0
        Orientation:
          Angle1 = 0.0
          Angle2 = 0.0
          Angle3 = 0.0
      Position[3]:
        Object = MyProduct
        Translation:
          X = 96.0
          Y = 0.0
          Z = 0.0
        Orientation:
          Angle1 = 0.0
          Angle2 = 0.0
          Angle3 = 0.0
      Position[4]:
        Object = MyProduct
        Translation:
          X = 144.0
          Y = 0.0
          Z = 0.0
        Orientation:
          Angle1 = 0.0
          Angle2 = 0.0
          Angle3 = 0.0
```

### Config_8.pickregister - 5APC3100_KBU1_000a/mappMotion/PnP_AddOn/Config_8.pickregister
```
Element gPickRegister (Type=pickregister)
  Type = LinearConveyor
    StandardFrameName = ConveyorPick
    Length = 300
    Width = 120
    Height = 10
    MotionSource = Axis
      AxisRef = gAxis_1
      MovementLimits = Internal
        Acceleration = Basic
  SceneViewerObject = Used
    VisualRepresentation = Conveyor belt
      Dimensions:
        Length = 610
        Width = 120
        Height = 50
      Translation:
        X = -150
        Y = 0.0
        Z = 0.0
      Orientation:
        Angle1 = 0.0
        Angle2 = 0.0
        Angle3 = 0.0
      Material = GreenMatte
    Content:
      Template[1]:
        VisualRepresentation:
          Size = 50.0
  Alarms = None
Element gPlaceRegister (Type=pickregister)
  Type = LinearConveyor
    StandardFrameName = ConveyorPlace
    Length = 205
    Width = 20
    Height = 10
    MaxItems = 5
    MotionSource = Axis
      AxisRef = gAxis_2
      AxisUsage = Passive
      MovementLimits = Internal
        Acceleration = Basic
  SceneViewerObject = Used
    VisualRepresentation = Cuboid
      Dimensions:
        Length = 215
        Width = 60
        Height = 50
      Translation:
        X = 0
        Y = -20
        Z = 0.0
      Orientation:
        Angle1 = 0.0
        Angle2 = 0.0
        Angle3 = 0.0
    Content:
      Template[1]:
        VisualRepresentation:
          Size = 50.0
  Alarms = None
```

### Config_9.pickcore - 5APC3100_KBU1_000a/mappMotion/PnP_AddOn/Config_9.pickcore
```
Element gPickCore_1 (Type=pickcore)
  AxesGroupRef = g4AxDeltaA
  Gripper = Standard
    Behavior:
      ProcessVariableName = ::PrgPickCor:Gripper
  Job[1]:
    JobName = PickToPlace
    Object = MyProduct
    InfeedRegister = gPickRegister
    OutfeedRegister = gPlaceRegister
    Movement = Basic
      PickOffsetZ = 50
      PickRounding = 30
      PlaceOffsetZ = 50
      PlaceRounding = 30
    Limits = NotUsed
  OperationMode[1]:
    Name = ConveyorToConveyor
    AssignedJob[1]:
      Name = ChaoticToLine
      Processing = FIFO
      JobExecBehav = WaitForPlaceHolder
    AssignedJob[2]:
      Name
      Processing = FIFO
      JobExecBehav = WaitForPlaceHolder
    AssignedJob[3]:
      Name
      Processing = FIFO
      JobExecBehav = WaitForPlaceHolder
    AssignedJob[4]:
      Name
      Processing = FIFO
      JobExecBehav = WaitForPlaceHolder
    AssignedJob[5]:
      Name
      Processing = FIFO
      JobExecBehav = WaitForPlaceHolder
    AssignedJob[6]:
      Name
      Processing = FIFO
      JobExecBehav = WaitForPlaceHolder
    AssignedJob[7]:
      Name
      Processing = FIFO
      JobExecBehav = WaitForPlaceHolder
    AssignedJob[8]:
      Name
      Processing = FIFO
      JobExecBehav = WaitForPlaceHolder
    AssignedJob[9]:
      Name
      Processing = FIFO
      JobExecBehav = WaitForPlaceHolder
    AssignedJob[10]:
      Name
      Processing = FIFO
      JobExecBehav = WaitForPlaceHolder
    IdleBehavior = StayFixedWaitingPosition
      Position:
        StandardFrameName = PnPWaitingPosition
        Translation:
          X = 0.0
          Y = 0.0
          Z = 0.0
        Orientation:
          Angle1 = 0.0
          Angle2 = 0.0
          Angle3 = 0.0
  Alarms = None
```

### Config.mppackmlcore - 5APC3100_KBU1_000a/mappServices/Config.mppackmlcore
```
Element gPackMLCore (Type=mppackmlcore)
  Modes:
    Mode[1]:
      ModeID = 1
      Name = Production
      State[1] = 0
      State[5] = 0
      State[10] = 0
      State[11] = 0
      State[12] = 0
      State[13] = 0
      State[14] = 0
      State[16] = 0
      State[17] = 0
```

### Config_11.mpalarmxcore - 5APC3100_KBU1_000a/mappServices/Config_11.mpalarmxcore
```
Element gAlarmXCore (Type=mpalarmxcore)
  mapp.AlarmX.Core.Configuration:
    [0]:
      Name = Alarm
      Message = Wystapil alarm
      Behavior = RateOfChangeMonitoring
        Monitoring:
          MonitoredPV = ::Alarmy:MpAlarmXCore_0.PendingAlarms
```

### Config_12.mpalarmxhistory - 5APC3100_KBU1_000a/mappServices/Config_12.mpalarmxhistory
```
Element gAlarmXHistory (Type=mpalarmxhistory)
  mapp.AlarmX.History:
    Auditing = MpAudit
    Scope = Branch
```

### Config_12.mpuserlogin - 5APC3100_KBU1_000a/mappServices/Config_12.mpuserlogin
```
Element gUserLogin (Type=mpuserlogin)
  Login:
    AutoLogout = 3600
```

### Config_13.mpuserx - 5APC3100_KBU1_000a/mappServices/Config_13.mpuserx
```
Element UserMgmtX (Type=mpuserx)
  Mgr:
    PasswordChangeInterval = 2592000
    PasswordExpirationNotification = 864000
    UserExpirationTime = 31536000
    PasswordChangeReq = TRUE
    PasswordCase = TRUE
    PasswordAlpha = TRUE
    PasswordLength = 3
    UserNameLength = 3
    PasswordHistory = 5
    LoginAttempts = 5
  ServerSettings:
    Server:
      AdditionalUserData:
        [0] = mail
        [1] = telephoneNumber
  Users:
    DefUser#1:
      id = Admin
      name = Admin
      lang = en
    DefUser#2:
      id = Anonymous
      name = Anonymous
      lang = en
    DefUser#3:
      id = Operator
      name = Operator
      lang = en
    DefUser#4:
      id = Maciek
      name = Maciek
      lang = en
  Groups:
    DefGroup#1:
      id = Administrators
      level = 100
      rights:
        [0] = FullAccess
        [1] = ViewOnly
        [2] = StartOnly
    DefGroup#2:
      id = Everyone
      level = 3
      rights:
        [0] = ViewOnly
    DefGroup#3:
      id = Operators
      level = 30
      rights:
        [0] = StartOnly
```

### Config_mS1.mpaudittrail - 5APC3100_KBU1_000a/mappServices/Config_mS1.mpaudittrail
```
Element gAuditTrail (Type=mpaudittrail)
  Audit:
    Events:
      [0] = 16
      [1] = 2
      [2] = 18
      [3] = 33
    TextSource:
      OutputFormat = [%[TIME=%c]] [%msg]
    Archive = On
    Export:
      Encrypt = FALSE
  Alarms = MpAlarmX
```

### viComp.visioncomponent - 5APC3100_KBU1_000a/mappVision/viComp.visioncomponent
```
Element gCamera (Type=visioncomponent)
  VisionApplicationReference = VisionMatching
```

### Config_1.axesgroup - CPU/mappMotion/4AxesDeltaA/Config_1.axesgroup
```
Element g4AxDeltaA (Type=axesgroup)
  Type = PathGenAxesGroup
    ProcessingTaskClass = 255
    License = 1
    PhysicalAxes:
      JointAxes:
        JointAxisAxisRefIsReadOnly = 0
        JointAxis[1]:
          Name = Q1
          AxisRef = gAxisQ1
        JointAxis[2]:
          Name = Q2
          AxisRef = gAxisQ2
        JointAxis[3]:
          Name = Q3
          AxisRef = gAxisQ3
        JointAxis[4]:
          Name = Q4
          AxisRef = gAxisQ4
    MechanicalSystem:
      MechSysRefIsReadOnly = 0
      MechSysRef = MechSys_4AxDeltaA
    BasicSettings:
      ModalDataBehaviour = ResetToDefault
      GeometryPlanning:
        TCPResolutionIsReadOnly = 0
        TCPResolution:
          LengthResolution = 0.001
          AngleResolution = 0.001
        Rounding:
          PathDistance = 0.0
          SymmetricRounding = Yes
          LastSegment = Half
          AvoidZeroCurvature = No
        RoundingMode = Standard
        MaxCornerDeviation = 0.0
        MaxTangentialTransitionDeviation = 0.0
        MaxRadiusDeviation = 0.001
        WorkingPlane = XY
      TrajectoryPlanningIsReadOnly = 0
      TrajectoryPlanning = Basic
        LimitCheckResolutionIsReadOnly = 0
        LimitCheckResolution = UserDefinedTime
          TimeIsReadOnly = 0
          Time = 0.005
        BufferTime = UserDefinedTime
          Time = 0.1
        BarrierParametrization = JointCoordinates
      Miscellaneous:
        NonMovementsLimit = NotUsed
        TimeStretchOverride:
          JerkSuppression = NotUsed
    StopReaction:
      AxisError:
        AxisReactionIsReadOnly = 0
    AxesGroupFeatures:
      FeatureRef[1] = Feature_Programs
      FeatureRef[2] = Feature_Jogging
      FeatureRef[3] = Feature_FrameHierarchy
      FeatureRef[4] = Feature_Tracking
      FeatureRef[5] = Feature_PathDefinition
    SceneObject:
      FileDevice = ComponentScenes
      FileNamePrefix = PathGen_
      FrameSize = 150
      FrameName = Invisible
      Positioner = NotUsed
      Object = Visible
      Boundaries = NotUsed
  Alarms = None
```

### Config_2.axis - CPU/mappMotion/4AxesDeltaA/Config_2.axis
```
Element gAxisQ1 (Type=axis)
  BaseTypeIsReadOnly = 0
  BaseType = RotaryBounded
    MeasurementUnitIsReadOnly = 0
    MeasurementUnit = 17476
    MeasurementResolutionIsReadOnly = 0
    MeasurementResolution = 0.01
    CountDirectionIsReadOnly = 0
    CountDirection = Standard
  MovementLimitsIsReadOnly = 0
  MovementLimits = InternalForPathControlledAxis
    Position:
      LowerLimitMin = -1.79769313486231E308
      UpperLimitMax = 1.79769313486231E308
      LowerLimit = -1000.0
      UpperLimit = 1000.0
    VelocityIsReadOnly = 0
    Velocity:
      VelocityMax = 3.4E38
      Velocity = 5000
    AccelerationIsReadOnly = 0
    Acceleration:
      AccelerationMax = 3.4E38
      Acceleration = 50000
    DecelerationIsReadOnly = 0
    Deceleration:
      DecelerationMax = 3.4E38
      Deceleration = 50000
    JerkIsReadOnly = 0
    Jerk = Basic
      JerkMax = 3.4E38
      Jerk = 500000
    TorqueIsInvisible = 0
    TorqueIsReadOnly = 0
  Alarms = None
Element gAxisQ2 (Type=axis)
  BaseTypeIsReadOnly = 0
  BaseType = RotaryBounded
    MeasurementUnitIsReadOnly = 0
    MeasurementUnit = 17476
    MeasurementResolutionIsReadOnly = 0
    MeasurementResolution = 0.01
    CountDirectionIsReadOnly = 0
    CountDirection = Standard
  MovementLimitsIsReadOnly = 0
  MovementLimits = InternalForPathControlledAxis
    Position:
      LowerLimitMin = -1.79769313486231E308
      UpperLimitMax = 1.79769313486231E308
      LowerLimit = -1000.0
      UpperLimit = 1000.0
    VelocityIsReadOnly = 0
    Velocity:
      VelocityMax = 3.4E38
      Velocity = 5000
    AccelerationIsReadOnly = 0
    Acceleration:
      AccelerationMax = 3.4E38
      Acceleration = 50000
    DecelerationIsReadOnly = 0
    Deceleration:
      DecelerationMax = 3.4E38
      Deceleration = 50000
    JerkIsReadOnly = 0
    Jerk = Basic
      JerkMax = 3.4E38
      Jerk = 500000
    TorqueIsInvisible = 0
    TorqueIsReadOnly = 0
  Alarms = None
Element gAxisQ3 (Type=axis)
  BaseTypeIsReadOnly = 0
  BaseType = RotaryBounded
    MeasurementUnitIsReadOnly = 0
    MeasurementUnit = 17476
    MeasurementResolutionIsReadOnly = 0
    MeasurementResolution = 0.01
    CountDirectionIsReadOnly = 0
    CountDirection = Standard
  MovementLimitsIsReadOnly = 0
  MovementLimits = InternalForPathControlledAxis
    Position:
      LowerLimitMin = -1.79769313486231E308
      UpperLimitMax = 1.79769313486231E308
      LowerLimit = -1000.0
      UpperLimit = 1000.0
    VelocityIsReadOnly = 0
    Velocity:
      VelocityMax = 3.4E38
      Velocity = 5000
    AccelerationIsReadOnly = 0
    Acceleration:
      AccelerationMax = 3.4E38
      Acceleration = 50000
    DecelerationIsReadOnly = 0
    Deceleration:
      DecelerationMax = 3.4E38
      Deceleration = 50000
    JerkIsReadOnly = 0
    Jerk = Basic
      JerkMax = 3.4E38
      Jerk = 500000
    TorqueIsInvisible = 0
    TorqueIsReadOnly = 0
  Alarms = None
Element gAxisQ4 (Type=axis)
  BaseTypeIsReadOnly = 0
  BaseType = Rotary
    MeasurementUnitIsReadOnly = 0
    MeasurementUnit = 17476
    MeasurementResolutionIsReadOnly = 0
    MeasurementResolution = 0.01
    CountDirectionIsReadOnly = 0
    CountDirection = Standard
  MovementLimitsIsReadOnly = 0
  MovementLimits = InternalForPathControlledAxis
    Position:
      LowerLimitMin = -1.79769313486231E308
      UpperLimitMax = 1.79769313486231E308
      LowerLimit = -1000.0
      UpperLimit = 1000.0
    VelocityIsReadOnly = 0
    Velocity:
      VelocityMax = 3.4E38
      Velocity = 5000
    AccelerationIsReadOnly = 0
    Acceleration:
      AccelerationMax = 3.4E38
      Acceleration = 50000
    DecelerationIsReadOnly = 0
    Deceleration:
      DecelerationMax = 3.4E38
      Deceleration = 50000
    JerkIsReadOnly = 0
    Jerk = Basic
      JerkMax = 3.4E38
      Jerk = 500000
    TorqueIsInvisible = 0
    TorqueIsReadOnly = 0
  Alarms = None
```

### Config_6.axesgroupfeature - CPU/mappMotion/PnP_AddOn/Config_6.axesgroupfeature
```
Element Feature_FrameHierarchy (Type=axesgroupfeature)
  Type = FrameHierarchy
    ModalDataBehaviour = UseAxesGroupSettings
    FrameHierarchy = Custom
      FramePropertyMapping:
        BCS = RoboBase
        PCS = ZeroPosPickConveyor
        SCS1
        SCS2
        SCS3
        SCS4
        SCS5
      MCS:
        Name = MachineBase
        Frame[1]:
          Name = RoboBase
          Type = StandardFrame
            Translation:
              X = 0.0
              Y = 0.0
              Z = 1000
            Orientation:
              Angle1 = 0.0
              Angle2 = 0.0
              Angle3 = 0.0
          Frame[1]:
            Name = ZeroPosPickConveyor
            Type = StandardFrame
              Translation:
                X = 0.0
                Y = 400
                Z = -1000
              Orientation:
                Angle1 = 0.0
                Angle2 = 0.0
                Angle3 = 0.0
Element Feature_Tracking (Type=axesgroupfeature)
  Type = Tracking
    ModalDataBehaviour = UseAxesGroupSettings
    SynchronisationGeometry = Basic
      CartesianRadius = 20.0
    TorqueLimitConsideration = Exact
Element Feature_PathDefinition (Type=axesgroupfeature)
  Type = PathDefinitions
    ModalDataBehaviour = UseAxesGroupSettings
    PathDefinition[1]:
      Name = Path1
      Type = CartesianPath
        CalculatedIn = PCS
      Limit = Internal
        Velocity = NotUsed
        Acceleration = NotUsed
        Deceleration = NotUsed
        Jerk = NotUsed
```

### Config_8.pickregister - CPU/mappMotion/PnP_AddOn/Config_8.pickregister
```
Element gPickRegister (Type=pickregister)
  Type = LinearConveyor
    StandardFrameName = ConveyorPick
    Length = 2000
    Width = 250
    MotionSource = Axis
      AxisRef = gAxis_1
      MovementLimits = UseAxisLimits
    SceneObject = Visible
      RegisterName = Visible
      Opacitiy = 0.45
      Dimensions = NotUsed
      ConveyorBelt = NotUsed
  SceneViewerSettings:
    FileDevice = CNC_PrgDir
    FileNamePrefix = PickRegister_
  Alarms = None
Element gPlaceRegister (Type=pickregister)
  Type = LinearConveyor
    StandardFrameName = ConveyorPlace
    Length = 2000
    Width = 250
    MotionSource = Axis
      AxisRef = gAxis_2
      MovementLimits = UseAxisLimits
    SceneObject = Visible
      RegisterName = Visible
      Opacitiy = 0.45
      Dimensions = NotUsed
      ConveyorBelt = NotUsed
  SceneViewerSettings:
    FileDevice = CNC_PrgDir
    FileNamePrefix = PlaceRegister_
  Alarms = None
```

### Config_1.axesgroup - PC/mappMotion/4AxesDeltaA/Config_1.axesgroup
```
Element g4AxDeltaA (Type=axesgroup)
  Type = PathGenAxesGroup
    ProcessingTaskClass = 255
    License = 1
    PhysicalAxes:
      JointAxes:
        JointAxisAxisRefIsReadOnly = 0
        JointAxis[1]:
          Name = Q1
          AxisRef = gAxisQ1
        JointAxis[2]:
          Name = Q2
          AxisRef = gAxisQ2
        JointAxis[3]:
          Name = Q3
          AxisRef = gAxisQ3
        JointAxis[4]:
          Name = Q4
          AxisRef = gAxisQ4
    MechanicalSystem:
      MechSysRefIsReadOnly = 0
      MechSysRef = MechSys_4AxDeltaA
    BasicSettings:
      ModalDataBehaviour = ResetToDefault
      GeometryPlanning:
        TCPResolutionIsReadOnly = 0
        TCPResolution:
          LengthResolution = 0.001
          AngleResolution = 0.001
        Rounding:
          PathDistance = 0.0
          SymmetricRounding = Yes
          LastSegment = Half
          AvoidZeroCurvature = No
        RoundingMode = Standard
        MaxCornerDeviation = 0.0
        MaxTangentialTransitionDeviation = 0.0
        MaxRadiusDeviation = 0.001
        WorkingPlane = XY
      TrajectoryPlanningIsReadOnly = 0
      TrajectoryPlanning = Basic
        LimitCheckResolutionIsReadOnly = 0
        LimitCheckResolution = UserDefinedTime
          TimeIsReadOnly = 0
          Time = 0.01
        BufferTime = UserDefinedTime
          Time = 0.1
        BarrierParametrization = JointCoordinates
        TorqueLimitConsideration = Exact
      Miscellaneous:
        NonMovementsLimit = NotUsed
        TimeStretchOverride:
          JerkSuppression = NotUsed
    StopReaction:
      AxisError:
        AxisReactionIsReadOnly = 0
    AxesGroupFeatures:
      FeatureRef[1] = Feature_Programs
      FeatureRef[2] = Feature_Jogging
  Alarms = None
```

### Config_1.axesgroup - X20CP1584/mappMotion/4AxesDeltaA/Config_1.axesgroup
```
Element g4AxDeltaA (Type=axesgroup)
  Type = PathGenAxesGroup
    ProcessingTaskClass = 255
    License = 1
    PhysicalAxes:
      JointAxes:
        JointAxisAxisRefIsReadOnly = 0
        JointAxis[1]:
          Name = Q1
          AxisRef = gAxisQ1
        JointAxis[2]:
          Name = Q2
          AxisRef = gAxisQ2
        JointAxis[3]:
          Name = Q3
          AxisRef = gAxisQ3
        JointAxis[4]:
          Name = Q4
          AxisRef = gAxisQ4
    MechanicalSystem:
      MechSysRefIsReadOnly = 0
      MechSysRef = MechSys_4AxDeltaA
    BasicSettings:
      ModalDataBehaviour = ResetToDefault
      GeometryPlanning:
        TCPResolutionIsReadOnly = 0
        TCPResolution:
          LengthResolution = 0.001
          AngleResolution = 0.001
        Rounding:
          PathDistance = 0.0
          SymmetricRounding = Yes
          LastSegment = Half
          AvoidZeroCurvature = No
        RoundingMode = Standard
        MaxCornerDeviation = 0.0
        MaxTangentialTransitionDeviation = 0.0
        MaxRadiusDeviation = 0.001
        WorkingPlane = XY
      TrajectoryPlanningIsReadOnly = 0
      TrajectoryPlanning = Basic
        LimitCheckResolutionIsReadOnly = 0
        LimitCheckResolution = UserDefinedTime
          TimeIsReadOnly = 0
          Time = 0.01
        BufferTime = UserDefinedTime
          Time = 0.1
        BarrierParametrization = JointCoordinates
        TorqueLimitConsideration = Exact
      Miscellaneous:
        NonMovementsLimit = NotUsed
        TimeStretchOverride:
          JerkSuppression = NotUsed
    StopReaction:
      AxisError:
        AxisReactionIsReadOnly = 0
    AxesGroupFeatures:
      FeatureRef[1] = Feature_FrameHierarchy
      FeatureRef[2] = Feature_Jogging
      FeatureRef[3] = Feature_PathDefinition
      FeatureRef[4] = Feature_Programs
      FeatureRef[5] = Feature_Tracking
  Alarms = None
```

### Config_3.mechanicalsystem - X20CP1584/mappMotion/4AxesDeltaA/Config_3.mechanicalsystem
```
Element MechSys_4AxDeltaA (Type=mechanicalsystem)
  TypeIsReadOnly = 0
  Type = Delta
    SubtypeIsReadOnly = 0
    Subtype = 4AxesDeltaA
      SceneViewerObject = Generic
      DescriptionIsReadOnly = 0
      Description = Standard
        Dimensions:
          BasePlatform:
            CenterIsReadOnly = 0
            Center:
              X = 0.0
              Y = 0.0
              Z = 0.0
            ArmLinkPointIsReadOnly = 0
            Arm1LinkPoint:
              Angle = 0.0
              Radius = 250.0
              Z = 0.0
            Arm2LinkPoint:
              Angle = 120.0
              Radius = 250.0
              Z = 0.0
            Arm3LinkPoint:
              Angle = 240.0
              Radius = 250.0
              Z = 0.0
          Arms:
            ArmIsReadOnly = 0
            Arm1:
              UpperArmLength = 600.0
              LowerArmLength = 900.0
            Arm2:
              UpperArmLength = 600.0
              LowerArmLength = 900.0
            Arm3:
              UpperArmLength = 600.0
              LowerArmLength = 900.0
            LowerArmPairDistance = 0.0
          EndEffectorPlatform:
            ArmLinkPointIsReadOnly = 0
            Arm1LinkPoint:
              Radius = 50.0
              Z = 0.0
            Arm2LinkPoint:
              Radius = 50.0
              Z = 0.0
            Arm3LinkPoint:
              Radius = 50.0
              Z = 0.0
            TranslationToFlangeIsReadOnly = 0
            TranslationToFlange:
              X = 0.0
              Y = 0.0
              Z = -150
        Offsets:
          JointAxisIsReadOnly = 0
          JointAxis[1] = 0.0
          JointAxis[2] = 0.0
          JointAxis[3] = 0.0
          JointAxis[4] = 0.0
        CountDirections:
          JointAxisIsReadOnly = 0
          JointAxis[1] = Standard
          JointAxis[2] = Standard
          JointAxis[3] = Standard
          JointAxis[4] = Standard
      CoordinatesNames = Default
        XCoordinateName = X
        YCoordinateName = Y
        ZCoordinateName = Z
        CCoordinateName = C
      TcpOrientation:
        Frames = Used
      WireFrameModelIsReadOnly = 0
      WireFrameModel = Standard
        UpperArm1IsReadOnly = 0
        UpperArm1 = ConnectionLine
          DistanceMin = -1.79769313486231E308
          DistanceMax = 1.79769313486231E308
          Distance = 0.0
        LowerArm1IsReadOnly = 0
        LowerArm1 = ConnectionLine
          DistanceMin = -1.79769313486231E308
          DistanceMax = 1.79769313486231E308
          Distance = 0.0
        UpperArm2IsReadOnly = 0
        UpperArm2 = ConnectionLine
          DistanceMin = -1.79769313486231E308
          DistanceMax = 1.79769313486231E308
          Distance = 0.0
        LowerArm2IsReadOnly = 0
        LowerArm2 = ConnectionLine
          DistanceMin = -1.79769313486231E308
          DistanceMax = 1.79769313486231E308
          Distance = 0.0
        UpperArm3IsReadOnly = 0
        UpperArm3 = ConnectionLine
          DistanceMin = -1.79769313486231E308
          DistanceMax = 1.79769313486231E308
          Distance = 0.0
        LowerArm3IsReadOnly = 0
        LowerArm3 = ConnectionLine
          DistanceMin = -1.79769313486231E308
          DistanceMax = 1.79769313486231E308
          Distance = 0.0
        EndEffectorPlatformToFlangeIsReadOnly = 0
        EndEffectorPlatformToFlange = ConnectionLine
          DistanceMin = -1.79769313486231E308
          DistanceMax = 1.79769313486231E308
          Distance = 0.0
        FlangeToTcp = ConnectionLine
          DistanceMin = -1.79769313486231E308
          DistanceMax = 1.79769313486231E308
          Distance = 0.0
      DynamicModel = DynParTable
        TableRef
      InternalDynamicModelIsReadOnly = 0
      InternalDynamicModel = NotUsed
      DynamicLimits = DynParTables
        GearboxLimitsTableRef
        CrossSectionLimitsTableRef
      InternalDynamicLimits = NotUsed
      CouplingsIsInvisible = 0
      JointAxesPositionLimits:
        JointAxisIsReadOnly = 0
        JointAxis[1] = UseAxisLimits
        JointAxis[2] = UseAxisLimits
        JointAxis[3] = UseAxisLimits
        JointAxis[4] = UseAxisLimits
      WorkingRangeIsReadOnly = 0
      WorkingRange = Standard
        BaseToTopIsReadOnly = 0
        BaseToTop = 400
        TopHeightIsReadOnly = 0
        TopHeight = 100
        MiddleHeightIsReadOnly = 0
        MiddleHeight = 400
        BottomHeightIsReadOnly = 0
        BottomHeight = 600
        TopRadiusIsReadOnly = 0
        TopRadius = 800
        MiddleRadiusIsReadOnly = 0
        MiddleRadius = 900
        BottomRadiusIsReadOnly = 0
        BottomRadius = 200
```

### Config_4.axesgroupfeature - X20CP1584/mappMotion/4AxesDeltaA/Config_4.axesgroupfeature
```
Element Feature_Programs (Type=axesgroupfeature)
  Type = Program
    ModalDataBehaviour = UseAxesGroupSettings
    InitialSettings:
      InterpolationTypes = LinearRapid
      PositionCoordinates = Absolute
      CircleCoordinates = Relative
      JACS_ACSProgramming = JACS
      ContourConnection = Inactive
      AccuracyHoldDelays = None
      ProgrammingUnits = UseAxesGroupSettings
      Feedrates:
        FeedPath = Standard
        FeedCharacteristic = StandardCharacteristic
        FeedType = Feedrate
        FeedReduction = Inactive
        FeedrateValue = 0.0
        InverseFeedrateValue = 0.0
        FeedratePerRevValue = 0.0
    DefaultLanguage = BRGCode
    Location = Default
      FileDevice = CNC_PrgDir
Element Feature_Jogging (Type=axesgroupfeature)
  Type = Jogging
Element Feature_Tracking (Type=axesgroupfeature)
  Type = Tracking
    ModalDataBehaviour = UseAxesGroupSettings
    SynchronisationGeometry = Basic
      CartesianRadius = 20
Element Feature_FrameHierarchy (Type=axesgroupfeature)
  Type = FrameHierarchy
    ModalDataBehaviour = UseAxesGroupSettings
    FrameHierarchy = Custom
      FramePropertyMapping:
        BCS = MachineFrame
        PCS = MachineFrame
        SCS1
        SCS2
        SCS3
        SCS4
        SCS5
Element Feature_PatchDefinition (Type=axesgroupfeature)
  Type = PathDefinitions
    ModalDataBehaviour = UseAxesGroupSettings
    PathDefinition[1]:
      Name = Path1
      Type = CartesianPath
        CalculatedIn = PCS
      Limit = Internal
        Velocity = NotUsed
        Acceleration = NotUsed
        Deceleration = NotUsed
        Jerk = NotUsed
```

## Logical view

Binary libraries used (declarations not repeated): McBase, MpBase, McTrkPath 5.24.1, CoTrace, AsZip, FileIO, runtime, McAcpAx, McAxis, McAxGroup 5.24.1, McPathGen 5.26.1, McProgInt 5.24.1, MpPick 5.26.1, McAcpTrak, MpAxis, MpCnc, MpRobotics 5.26.1, MpTool, sys_lib, McAcpPar, McDS402Ax 5.24.1, McPureVAx, McStpAx 5.26.1, MpServer, AsIODiag, MpAudit 5.24.2, MpPackML 5.24.2, AsARCfg, powerlnk, AsEPL, AsIO, DataObj, MpAlarmX 5.24.2, standard, MpUser 5.24.2, ViBase 5.24.1, MpWebXs 5.24.2, AsArSdm, asstring, AsHttp, UserLib, McPathGen, McTrkPath, MpRobotics 5.24.1

### Global.var - Global variables
```iecst
VAR CONSTANT
	P1 : McPointType := (Pos:=(X:=0,Y:=0,Z:=-650));
	P2 : McPointType := (Pos:=(X:=-50,Y:=-20,Z:=-600));
	P0 : McPointType := (Pos:=(X:=0,Y:=0,Z:=-560));
	P3 : McPointType := (Pos:=(X:=50,Y:=20,Z:=-540));
END_VAR
VAR
	TablePosition : LREAL := 5;
	ProgramPickExecuteBool : BOOL;
	AbortExecute : BOOL;
	StopExecute : BOOL;
	StopExecutedPick : BOOL;
	AbortExecutedPick : BOOL;
	StopExecutedPickCore : BOOL;
	StopExecutedPlace : BOOL;
	ResetExecutePickCore : BOOL;
	gTokenStartPosY : USINT;
	CmdStart : BOOL := FALSE; (*Set = 1 to start the process*)
	gIsCameraActive : BOOL;
	ConvVelocityDegrees : REAL;
	gDeleteObjects : BOOL;
	gManualHoming : BOOL;
	gManualMode : BOOL;
	gIsConvHomed : BOOL;
	gMakeToken : BOOL;
	ResetExecutedPickCore : BOOL;
	gTokenOnConv : BOOL;
	gToken_Y : REAL;
	gToken_X : REAL;
	gAbort : BOOL := FALSE;
	ClearingExecute : BOOL;
	ClearingExecutedPick : BOOL;
	ClearingExecutedPickCore : BOOL;
	ClearingExecutedPlace : BOOL;
END_VAR
```

- mCoWebServ4.mcowebservercfg (not shown)

### Robotic.st
```iecst
PROGRAM _MAIN
	Feedrate(5000);   //move with reduced speed
	MoveJ(P1);        //move system to point P1
	MoveJ(P2);        //move system to point P2

	WaitTime(3);        //wait for 3 seconds

	MoveJ(P0);        //move back to origin position
	END_PROGRAM
```

### PrgGlobal.var - Pick and place global variables
```iecst
VAR
	ReadyMechanics : BOOL := FALSE;
	ReadyPickCore : BOOL := FALSE;
	ReadyPickReg : BOOL := FALSE;
	ReadyPlaceReg : BOOL := FALSE;
	ReadyToStart : BOOL := FALSE;
	PickConveyorPosition : LREAL;
	PickConveyorLength : LREAL := 600; (*must be the same as pick conveyor length in MpPick configuration*)
	PlaceConveyorPosition : LREAL;
	PlaceConveyorLength : LREAL := 205; (*must be the same as place conveyor length in MpPick configuration*)
	gContainerInfo : ARRAY[0..3] OF MpPickObjPosInfoType;
	gTokenNumber : {REDUND_UNREPLICABLE} UDINT := 0;
	gMpDelta4AxisEnable : BOOL;
	gMpDelta4AxisJog : BOOL;
	DeltaParamConnections : MpDelta4AxisParType;
	gTcpPositionX : LREAL;
	gTcpPositionY : LREAL;
	gTcpPositionZ : LREAL;
END_VAR
```

### Program Logical/PickAndPlace/PrgPickCore (IEC) - PickCore process handling

#### Main.st
```iecst
PROGRAM _INIT

    PC_Step := PC_ENABLE_PICK_CORE;
    Gripper := FALSE;

END_PROGRAM

PROGRAM _CYCLIC

	IF NOT(gManualMode) THEN

	    CASE PC_Step OF

	        (* Enable the PickCore *)
			PC_ENABLE_PICK_CORE:
				IF NOT AbortExecute AND NOT StopExecute AND NOT MpPickCore_0.Error THEN
					StopExecutedPickCore := FALSE;
					MpPickCore_0.ProcessStop := FALSE;
					PC_Step := PC_WAIT_ENABLE_PICK_CORE;
					ClearingExecutedPickCore := FALSE;
					MpPickCore_0.ErrorReset := FALSE;
				END_IF

			PC_WAIT_ENABLE_PICK_CORE:
				MpPickCore_0.Enable := TRUE;
	            IF MpPickCore_0.Active THEN
	                PC_Step := PC_ENABLE_CORE_PROCESS;

				ELSIF MpPickCore_0.Error THEN
					LastStep := PC_Step;
	                PC_Step  := PC_ERROR;

				END_IF;

	        PC_ENABLE_CORE_PROCESS:
	            MpPickCore_0.ProcessEnable := TRUE;
	            PC_Step := PC_WAIT_ENABLE_CORE_PROCESS;

	        PC_WAIT_ENABLE_CORE_PROCESS:
	            IF MpPickCore_0.ProcessActive THEN
	                PC_Step := PC_READY_TO_START;

	            ELSIF MpPickCore_0.Error THEN
					LastStep := PC_Step;
	                PC_Step  := PC_ERROR;

	            END_IF

	        PC_READY_TO_START:
	            ReadyPickCore := TRUE;

	            IF CmdStart THEN
	                MpPickCore_0.Parameters.OperationMode := 'ConveyorToConveyor';  //ZMIENIONE NA CZAS TESTOW!!!!!!
				    MpPickCore_0.ProcessStart := TRUE;
	                PC_Step := PC_WAIT_START_CORE_PROCESS;
	            END_IF

	        PC_WAIT_START_CORE_PROCESS:
				IF MpPickCore_0.ProcessRunning THEN
	                PC_Step := PC_STARTED;

				ELSIF MpPickCore_0.Error THEN
					LastStep := PC_Step;
	                PC_Step  := PC_ERROR;

				END_IF;

	        PC_STARTED:
	            (* Nothing to do here *)
	            IF MpPickCore_0.Error THEN
					LastStep := PC_Step;
	                PC_Step  := PC_ERROR;
				END_IF;

	        PC_ERROR:
	            Error := TRUE;
	            ReadyPickCore := FALSE;

		END_CASE

		IF StopExecute THEN
			PC_Step := PC_ENABLE_PICK_CORE;
			ReadyPickCore := FALSE;
			StopExecutedPickCore := TRUE;
		ELSIF AbortExecute THEN
			MpPickCore_0.ProcessStop := TRUE;
			PC_Step := PC_ENABLE_PICK_CORE;
			ReadyPickCore := FALSE;
			StopExecutedPickCore := TRUE;
		END_IF

		IF ResetExecutePickCore THEN
			MpPickCore_0.ProcessStop := FALSE;
			MpPickCore_0.ProcessStart := FALSE;
			PC_Step := PC_ENABLE_PICK_CORE;
			ResetExecutedPickCore := TRUE;
			Error := FALSE;
		END_IF

		IF ClearingExecute THEN
			MpPickCore_0.ErrorReset := TRUE;
			ClearingExecutedPickCore := TRUE;
		END_IF

	    (* Call FBs *)
	    MpPickCore_0.MpLink := ADR(gPickCore_1);
		MpPickCore_0();

		//ELSE MpPickCore_0.Enable := FALSE;
	END_IF

END_PROGRAM
```

### Program Logical/PickAndPlace/PrgPick (IEC) - Pick the products

#### Variables.var
```iecst
VAR
	C_Step : ConvStepEnum;
	LastStep : ConvStepEnum;
	Error : BOOL;
	ProductSpacing : LREAL;
	LastProductConveyorPosition : LREAL;
	ElapsedDistance : LREAL;
	OldMakeToken : BOOL;
END_VAR
(*  *)
(*Functionblocks*)
VAR
	MpPickRegister_0 : MpPickRegister;
	MpPickRegCreateProduct : MpPickRegCreateObject;
END_VAR
```

#### Main.st
```iecst
PROGRAM _INIT

	C_Step := C_WAIT_ENABLE;
	Error := FALSE;

	ProductSpacing := 120; // distance between two consecutive products

END_PROGRAM

PROGRAM _CYCLIC

	IF NOT(gManualMode) THEN

	CASE C_Step OF
		C_WAIT_ENABLE:
			LastStep := C_WAIT_ENABLE;
			IF NOT AbortExecute AND NOT StopExecute AND NOT MpPickRegister_0.Error THEN
				C_Step   := C_ENABLE_REGISTER_FB;
				StopExecutedPick := FALSE;
				ClearingExecutedPick := FALSE;
				MpPickRegister_0.ErrorReset := FALSE;
			END_IF

			(* Pick-and-Place register handling for Picking conveyor *)
		C_ENABLE_REGISTER_FB:
			MpPickRegister_0.Enable := TRUE;
			C_Step := C_WAIT_ENABLE_REGISTER_FB;

		C_WAIT_ENABLE_REGISTER_FB:
			IF MpPickRegister_0.Active THEN
				C_Step := C_ENABLE_REGISTER;
			ELSIF MpPickRegister_0.Error THEN
				LastStep := C_Step;
				C_Step   := C_ERROR;
			END_IF;

		C_ENABLE_REGISTER:
			MpPickRegister_0.RegisterEnable := TRUE;
			C_Step := C_WAIT_ENABLE_REGISTER;

		C_WAIT_ENABLE_REGISTER:
			IF MpPickRegister_0.RegisterActive THEN
				C_Step := C_ENABLE_ADD_REGISTER_FBS;
			ELSIF MpPickRegister_0.Error THEN
				LastStep := C_Step;
				C_Step   := C_ERROR;
			END_IF;

		C_ENABLE_ADD_REGISTER_FBS:
			MpPickRegCreateProduct.Enable := TRUE;
			C_Step := C_WAIT_ENABLE_ADD_REGISTER_FBS;

		C_WAIT_ENABLE_ADD_REGISTER_FBS:
			IF MpPickRegCreateProduct.Active THEN
				C_Step := C_WAIT_START_PROCESS;
			ELSIF MpPickRegCreateProduct.Error THEN
				LastStep := C_Step;
				C_Step   := C_ERROR;
			END_IF;

		C_WAIT_START_PROCESS: // waits user start command and conveyor moving
			ReadyPickReg := TRUE;
			IF CmdStart AND ReadyToStart AND (PickConveyorPosition > 0) THEN
				C_Step := C_PROCESSING;
			END_IF;

		C_PROCESSING: (* now create products on moving conveyor for picking *)

			ElapsedDistance := DistanceOverPeriod(PickConveyorPosition, LastProductConveyorPosition, PickConveyorLength);

			IF EDGEPOS(gMakeToken) THEN

				MpPickRegCreateProduct.Parameters.LatchedConveyor.Position:= PickConveyorPosition;
				MpPickRegCreateProduct.Parameters.Mode := mpPICK_CREATE_SINGLEITEM;
				MpPickRegCreateProduct.Parameters.ObjectTypeName := 'MyProduct';
				MpPickRegCreateProduct.Parameters.Translation.X  := gToken_Y;
				MpPickRegCreateProduct.Parameters.Translation.Y  := gToken_X; // in the middle of conveyor width
					MpPickRegCreateProduct.Parameters.Translation.Z  := 2;
					MpPickRegCreateProduct.Create := TRUE;
					gTokenOnConv := TRUE;
				gMakeToken := FALSE;

				LastProductConveyorPosition := MpPickRegCreateProduct.Parameters.LatchedConveyor.Position;
			ELSE
				MpPickRegCreateProduct.Create := FALSE;
			END_IF

			IF MpPickRegCreateProduct.Error THEN
				LastStep := C_Step;
				C_Step   := C_ERROR;
			END_IF;

		C_ERROR:
			Error := TRUE;
			ReadyPickReg := FALSE;

	END_CASE

	IF StopExecute THEN
		C_Step := C_WAIT_ENABLE;
		ReadyPickReg := FALSE;
		StopExecutedPick := TRUE;
	END_IF

	IF MpPickRegCreateProduct.Error OR MpPickRegister_0.Error THEN
		gAbort := TRUE;
	END_IF

	IF AbortExecute THEN
		ReadyPickReg := FALSE;
		StopExecutedPick := TRUE;
		MpPickRegCreateProduct.Enable := FALSE;
		MpPickRegister_0.RegisterEnable := FALSE;
		MpPickRegister_0.Enable := FALSE;
	END_IF

	IF ClearingExecute THEN
		C_Step := C_WAIT_ENABLE;
		MpPickRegister_0.ErrorReset := TRUE;
		ClearingExecutedPick := TRUE;
	END_IF

	(* FB calls *)
	MpPickRegister_0.MpLink := ADR(gPickRegister);
	MpPickRegister_0();

	MpPickRegCreateProduct.MpLink := ADR(gPickRegister);
	MpPickRegCreateProduct();

	END_IF

END_PROGRAM
```

### Program Logical/PickAndPlace/MainProg (IEC)

#### Main.st - Init, cyclic, exit code
```iecst
PROGRAM _INIT
	MainInitAction;

END_PROGRAM

PROGRAM _CYCLIC

	//Configuring PackML
	MpPackCyclicAction;

	PackMLCurrentState := MpPackMLStateCurrent(gPackMLCore);

	// State machine in PackML standard
	CASE PackMLCurrentState OF
		mpPACKML_STATE_UNDEFINED:

			PackMLCurrentStateString := 'Undefined';
		//State in which pcoess is being stopped slowly
		mpPACKML_STATE_STOPPING:

			PackMLCurrentStateString := 'Stopping';
			MpAxisBasic_0.MoveVelocity := FALSE;
			MpAxisBasic_1.MoveVelocity := FALSE;

			StopExecute := TRUE;
			CmdStart := FALSE;
			IF StopExecutedPick AND StopExecutedPickCore AND StopExecutedPlace THEN
				ReadyMechanics := FALSE;
				MpPackMLStateComplete(gPackMLCore,1);
			END_IF

		// Program is stopped and waiting for reset command
		mpPACKML_STATE_STOPPED:
			MpAxisBasic_0.ErrorReset := FALSE;
			MpDelta4Axis_0.ErrorReset := FALSE;
			ClearingExecute := FALSE;
			PackMLCurrentStateString := 'Stopped';
			MpPackMLMode_0.Clear := FALSE;
			MpPackMLMode_0.Stop := FALSE;
			StopExecute := FALSE;
			RES_Step := HOMING_DELTA;

		// Program parameters are reseting in this state
		mpPACKML_STATE_RESETTING:
			PackMLCurrentStateString := 'Resetting';
			MpPackMLMode_0.Reset := FALSE;
			gDeleteObjects := TRUE;
			ResetExecutePickCore := TRUE;
			IF ResetExecutedPickCore THEN
				ResetingAction;
			END_IF

		// Idle state - watiting for START command
		mpPACKML_STATE_IDLE:
			PackMLCurrentStateString := 'Idle';
			gDeleteObjects := FALSE;
			ResetExecutePickCore := FALSE;
			ResetExecutedPickCore := FALSE;
			ReadyMechanics := TRUE;
			IF CmdStart AND ReadyToStart THEN
				MpPackMLMode_0.Start := TRUE;
			END_IF;

		// Starting state - conveyor start
		mpPACKML_STATE_STARTING:
			PackMLCurrentStateString := 'Starting';
			MpPackMLMode_0.Start := FALSE;
			IF NOT(gManualMode) THEN
				MpAxisBasic_0.MoveVelocity := TRUE;
				MpAxisBasic_1.MoveVelocity := TRUE;

				IF MpAxisBasic_0.Info.PLCopenState = mcAXIS_CONTINUOUS_MOTION THEN
					ProgramPickExecuteBool := TRUE;		// condition in Pick program
					MpPackMLStateComplete(gPackMLCore,1);
				END_IF
			END_IF

		mpPACKML_STATE_EXECUTE:
			IF NOT MpAxisBasic_0.PowerOn OR NOT MpDelta4Axis_0.PowerOn THEN
				gAbort := TRUE;
			END_IF
			PackMLCurrentStateString := 'Execute';
		// aborting -> when imidiate stop is in use
		mpPACKML_STATE_ABORTING:
			PackMLCurrentStateString := 'Aborting';
			AbortingAction;

		// Program is aborted. powers are shut down - waiting for cleaning command
		mpPACKML_STATE_ABORTED:
			PackMLCurrentStateString := 'Aborted';
			AbortExecute := FALSE;
			gAbort := FALSE;

			//Clearing alarms/bugs/warnings
		mpPACKML_STATE_CLEARING:
			ClearingExecute := TRUE;
			PackMLCurrentStateString := 'Clearing';
			IF ClearingExecutedPick
				AND ClearingExecutedPickCore
				AND ClearingExecutedPlace THEN
				MpAxisBasic_0.ErrorReset := TRUE;
				MpDelta4Axis_0.ErrorReset := TRUE;
				MpPackMLStateComplete(gPackMLCore,1);
			END_IF

	END_CASE;
	MpPackMLMode_0.Abort := gAbort;
	ReadyToStart := ReadyMechanics AND ReadyPickReg AND ReadyPlaceReg AND ReadyPickCore;

	//Conveyor homing information for camera
	IF MpAxisBasic_0.IsHomed THEN
		gIsConvHomed := TRUE;
   ELSE
		gIsConvHomed := FALSE;
	END_IF

	//Manual move configuration
	CheckManualAction;

	//MpPack init
	MpPackMLMode_0();
	MpPackMLCore_0();

	//All axis configuration -mplink -config -init
	AxisConfigAction;
    ConvVelocityDegrees:=MpAxisBasic_0.Velocity;
	//Updating both conveyors position
	PickConveyorPosition  := MpAxisBasic_0.Position;
	PlaceConveyorPosition := MpAxisBasic_1.Position;

END_PROGRAM

PROGRAM _EXIT
	(* Insert code here *)

END_PROGRAM
```

#### Types.typ - Local data types
```iecst
TYPE
	PML_CommandType : 	STRUCT  (*Commands structure*)
		UnitMode : DINT; (*Unit Mode target [Covered by MpPackMLCore PackTags]*)
		UnitModeChangeRequest : BOOL; (*Request Unit Mode change [Covered by MpPackMLCore PackTags]*)
		MachSpeed : REAL; (*Current machine speed [Primary packages/minute]*)
		MaterialInterlock : ARRAY[0..31]OF BOOL; (*Materials ready: MaterialInterlocks describes the status of the materials that are ready for processing*)
		CntrlCmd : DINT; (*Control Command [0=Undefined, 1=Reset, 2=Start, 3=Stop, 4=Hold, 5=Unhold, 6=Suspend, 7=Unsuspend, 8=Abort, 9=Clear] [Covered by MpPackMLCore PackTags]*)
		CmdChangeRequest : BOOL; (*State change request [Covered by MpPackMLCore PackTags]*)
		RemoteInterface : ARRAY[0..4]OF PML_RemoteInterfaceType; (*Upstream or downstream machine*)
		Parameter : ARRAY[0..4]OF PML_ParameterType; (*Parameter tags are associated to the end user supervisory interface*)
		Product : ARRAY[0..4]OF PML_ProductType; (*Product data type can be used for defining product and product processing parameter variables*)
	END_STRUCT;
	PML_StatusType : 	STRUCT  (*Status structure*)
		UnitModeCurrent : DINT; (*Unit Mode in current use [0=Invalid, 1=Production, 2=Maintenance, 3=Manual, 4-31=User definable) [Covered by MpPackMLCore PackTags]*)
		UnitModeRequested : BOOL; (*Requested Unit Mode change [Covered by MpPackMLCore PackTags]*)
		UnitModeChangeInProcess : BOOL; (*Requested Unit Mode change is in process [Covered by MpPackMLCore PackTags]*)
		StateCurrent : DINT; (*Current State Number [0=Undefined, 1=Clearing, 2=Stopped, 3=Starting, 4=Idle, 5=Suspended, 6=Execute, 7=Stopping, 8=Aborting, 9=Aborted, 10=Holding, 11=Held, 12=Unholding, 13=Suspending, 14=Unsuspending, 15=Resetting, 16=Completing, 17=Complete] [Covered by MpPackMLCore PackTags]*)
		StateRequested : DINT; (*Target State [0=Undefined, 1=Clearing, 2=Stopped, 3=Starting, 4=Idle, 5=Suspended, 6=Execute, 7=Stopping, 8=Aborting, 9=Aborted, 10=Holding, 11=Held, 12=Unholding, 13=Suspending, 14=Unsuspending, 15=Resetting, 16=Completing, 17=Complete]*)
		StateChangeInProcess : BOOL; (*State Change is in process [Covered by MpPackMLCore PackTags]*)
		MachSpeed : REAL; (*Current Machine Speed setpoint [Primary packages/minute]*)
		CurMachSpeed : REAL; (*Current Machine Speed real [Primary packages/minute]*)
		MaterialInterlock : ARRAY[0..31]OF BOOL; (*Materials ready: MaterialInterlocks describes the status of the materials that are ready for processing*)
		EquipmentInterlock : PML_EquipmentInterlockType; (*UpStream or downstream status*)
		RemoteInterface : ARRAY[0..4]OF PML_RemoteInterfaceType; (*Upstream or downstream machine*)
		Parameter : ARRAY[0..4]OF PML_ParameterType; (*Parameter tags are associated to the end user supervisory interface*)
		Product : ARRAY[0..4]OF PML_ProductType; (*Product data type can be used for displaying product and product processing parameter variables*)
	END_STRUCT;
	PML_AdminType : 	STRUCT  (*Administration structure*)
		Parameter : ARRAY[0..4]OF PML_ParameterType; (*Parameter tags associated to the local Interface are typically used for as parameters that are displayed or used on the unit locally, for example from an HMI*)
		Alarm : ARRAY[0..4]OF PML_AlarmType; (*Array of given size for machine fault number and messaging*)
		AlarmExtent : DINT; (*Extent of alarm array: the alarm extent is associated with the maximum number of alarms needed for the machine annunciation or reporting*)
		AlarmHistory : ARRAY[0..4]OF PML_AlarmType; (*Array of given size for machine fault number and messaging history*)
		AlarmHistoryExtent : DINT; (*Extent of alarm history array: the alarm history extent is associated with the maximum number of alarms needed to be archived or tagged as alarm history for the machine*)
		StopReason : PML_AlarmType; (*Machine stop reason is typically used for  First Out Fault  reporting and other stoppage events. The stop reason is the first event captured during an abort, held, suspended or stop event*)
		StopReasonExtent : DINT; (*Extent of stop reason array: the stop reason extent is associated with the maximum number of stop reasons needed to be archived or tagged as stop reasons for the machine*)
		Warning : PML_AlarmType; (*Machine warning are for general events that do not cause the machine to stop, but may require operator action as a stoppage may be imminent*)
		WarningExtent : DINT; (*The warning extent is associated with the maximum number of warnings needed to be archived or tagged as warnings for the machine*)
		ModeCurrentTime : ARRAY[0..31]OF DINT; (*Current amount of time (in sec) in any defined unit mode [Covered by MpPackMLCore PackTags]*)
		ModeCumulativeTime : ARRAY[0..31]OF DINT; (*Cumulative amount of time (in sec) in any defined unit mode [Covered by MpPackMLCore PackTags]*)
		StateCurrentTime : ARRAY[0..31]OF PML_ModeStateType; (*Current amount of time (in sec) in any defined state in any particular mode [Covered by MpPackMLCore PackTags]*)
		StateCumulativeTime : ARRAY[0..31]OF PML_ModeStateType; (*Cumulative amount of time (in sec) in any defined state in any particular mode since the last timer and counter reset was executed [Covered by MpPackMLCore PackTags]*)
		ProdConsumedCount : ARRAY[0..4]OF PML_ProdCountType; (*Material used / consumed in the production machine*)
		ProdProcessedCount : ARRAY[0..4]OF PML_ProdCountType; (*Number of products processed by the production machine*)
		ProdDefectiveCount : ARRAY[0..4]OF PML_ProdCountType; (*Product that is marked as defective in the production machine*)
		AccTimeSinceReset : DINT; (*Accumulative time since last reset [Covered by MpPackMLCore PackTags]*)
		MachDesignSpeed : REAL; (*Machine design speed [Primary Packages/minute]: maximum design speed of the machine in primary packages per minute for the package configuration being run*)
		StatesDisabled : DINT; (*States 1 to 17 of the PackML State Model can be disabled by turning on the corresponding bit in the INT.  Note that some state transition rules may over-ride the disable bits.  For Example, if HOLDING is not disabled, then HELD cannot be disabled*)
		PLCDateTime : PML_DateTimeType; (*Current Date and Time of the Programmable Logic Controller [Covered by MpPackMLCore PackTags]*)
	END_STRUCT;
	PML_RemoteInterfaceType : 	STRUCT  (*Upstream or downstream machine*)
		Number : DINT; (*Identification number of upstream or downstream unit machine*)
		ControlCmdNumber : DINT; (*Control command for upstream or downstream machine*)
		CmdValue : DINT; (*Control command value associated ControlCmdNumber*)
		Parameter : ARRAY[0..4]OF PML_ParameterType; (*Parameter tags associated to commanded remote interface*)
	END_STRUCT;
	PML_ParameterType : 	STRUCT  (*Parameter structure*)
		ID : DINT; (*ID value of Parameter*)
		Name : STRING[50]; (*String value assigned to Parameter*)
		Unit : STRING[5]; (*String value of Parameter units*)
		Value : REAL; (*Numeric value of Parameter*)
	END_STRUCT;
	PML_ProductType : 	STRUCT  (*Product structure*)
		ProductID : DINT; (*Structured array of Product ID#*)
		ProcessVariables : ARRAY[0..4]OF PML_ParameterType; (*Array of  data type Descriptor*)
		Ingredients : ARRAY[0..4]OF PML_IngredientsType; (*Structured Array for Ingredient Identification Parameters*)
	END_STRUCT;
	PML_AlarmType : 	STRUCT  (*Alarm structure*)
		Trigger : BOOL; (*Alarm Trigger should be turned on only when the alarm is currently active*)
		ID : DINT; (*Alarm message identification number *)
		Value : DINT; (*Alarm message number *)
		Message : STRING[80]; (*Alarm message*)
		Category : DINT; (*Alarm category: Category is used to identity what type of alarm has occurred (e.g. electrical, mechanical, materials, utilities, etc.)*)
		AlmDateTime : PML_DateTimeType; (*Structure of date and time in the alarm array to detail the date and time the alarm occurred*)
		AckDateTime : PML_DateTimeType; (*Structure of date and time in the alarm array to detail the date and time the alarm was acknowledged*)
	END_STRUCT;
	PML_IngredientsType : 	STRUCT  (*Ingredients structure*)
		IngredientID : DINT; (*The IngredientID is an arbitrary number associated with the raw material, or ingredient for a particular product number*)
		Parameter : ARRAY[0..4]OF PML_ParameterType; (*This array or structures is used for parameters associated with a particular ingredient or raw material used the processing of a particular product number*)
	END_STRUCT;
	PML_ProdCountType : 	STRUCT  (*Product count structure*)
		ID : DINT; (*This is the arbitrary (user defined) ID value of the consumed production material*)
		Name : STRING[80]; (*The name is used to literally describe the material ID, and its associated material*)
		Unit : STRING[5]; (*The unit tag is used to describe the names associated with a specific material used by the machine*)
		Count : DINT; (*The count value is used as a variable for displaying information about the amount of consumed production material*)
		AccCount : DINT; (*The accumulative count value is used as a variable for displaying information about the total amount of consumed production material*)
	END_STRUCT;
	PML_ModeStateType : 	STRUCT  (*Mode / State structure*)
		State : ARRAY[0..17]OF DINT; (*State inside each mode*)
	END_STRUCT;
	PML_EquipmentInterlockType : 	STRUCT  (*UpStream or downstream status*)
		Blocked : BOOL; (*This bit indicates that a downstream system is not able to accept product*)
		Starved : BOOL; (*This bit indicates that an upstream system is not able to supply product*)
	END_STRUCT;
	PML_DateTimeType : 	STRUCT  (*Date and time format*)
		Year : DINT; (*Date format: Year*)
		Month : DINT; (*Date format: Month*)
		Day : DINT; (*Date format: Day*)
		Hour : DINT; (*Time format: hours (24 hours format)*)
		Min : DINT; (*Time format: minutes*)
		Sec : DINT; (*Time format: seconds*)
		uSec : DINT; (*Time format: microseconds*)
	END_STRUCT;
	RES_StepType :
		(
		HOMING_DELTA,
		ACTIVATE_AXIS,
		HOMING_AXIS,
		COMPLETE_STATE
		);
END_TYPE
```

#### Variables.var - Local variables
```iecst
VAR
	MpPackMLCore_0 : MpPackMLCore;
	MpPackMLMode_0 : MpPackMLMode;
	homingModeQ1 : MpAxisBasicParType;
	MpDelta4Axis_0 : MpDelta4Axis;
	DeltaParameters : MpDelta4AxisParType;
	MpAxisBasic_0 : MpAxisBasic;
	AxisParameters_0 : MpAxisBasicParType;
	MpAxisBasic_1 : MpAxisBasic;
	AxisParameters_1 : MpAxisBasicParType;
	MpAxisBasic_Q1 : MpAxisBasic;
	MpAxisBasic_Q2 : MpAxisBasic;
	MpAxisBasic_Q3 : MpAxisBasic;
	Delta : MpAxisBasic;
	MpAxisBasic_Q4 : MpAxisBasic;
	homingModeQ3 : MpAxisBasicParType;
	homingModeQ4 : MpAxisBasicParType;
	homingModeQ2 : MpAxisBasicParType;
	PackMLCurrentState : MpPackMLStateEnum;
	RES_Step : RES_StepType;
	PackMLCurrentStateString : STRING[80];
END_VAR
```

#### ActionReseting.st
```iecst
ACTION ResetingAction:

	CASE RES_Step OF
		HOMING_DELTA:
			MpDelta4Axis_0.Home := TRUE;
			IF MpDelta4Axis_0.IsHomed THEN
				MpDelta4Axis_0.Home := FALSE;
				RES_Step := ACTIVATE_AXIS;
			END_IF

		ACTIVATE_AXIS:
			IF MpAxisBasic_0.Active AND MpDelta4Axis_0.Active THEN
				MpDelta4Axis_0.Power := TRUE;
				MpAxisBasic_0.Power := TRUE;
				MpAxisBasic_1.Power := TRUE; // axis not used, do not worry
				IF MpAxisBasic_0.PowerOn AND MpDelta4Axis_0.PowerOn THEN
					MpAxisBasic_0.MoveVelocity := FALSE;
					RES_Step := HOMING_AXIS;
				END_IF

			END_IF

		HOMING_AXIS:
			IF MpAxisBasic_0.PowerOn THEN
				MpAxisBasic_0.Home := TRUE;
				MpAxisBasic_1.Home := TRUE; // axis not used, do not worry
			END_IF;
			IF MpAxisBasic_0.IsHomed THEN
				MpAxisBasic_0.Home := FALSE;
				MpAxisBasic_1.Home := FALSE; // axis not used, do not worry
				RES_Step := COMPLETE_STATE;
			END_IF
		COMPLETE_STATE:
			MpPackMLStateComplete(gPackMLCore,1);

		END_CASE;
END_ACTION
```

#### CheckManual.st
```iecst
ACTION CheckManualAction:

	gTcpPositionX := MpDelta4Axis_0.X;
	gTcpPositionY := MpDelta4Axis_0.Y;
	gTcpPositionZ := MpDelta4Axis_0.Z;

	IF gManualMode THEN
		DeltaParameters.Jog.Velocity[0] := DeltaParamConnections.Jog.Velocity[0];
		DeltaParameters.Jog.Velocity[1] := DeltaParamConnections.Jog.Velocity[1];
		DeltaParameters.Jog.Velocity[2] := DeltaParamConnections.Jog.Velocity[2];
		DeltaParameters.ManualMoveType := DeltaParamConnections.ManualMoveType;
		DeltaParameters.Jog.CoordSystem := DeltaParamConnections.Jog.CoordSystem;
		DeltaParameters.CoordSystem := DeltaParamConnections.CoordSystem;
		MpDelta4Axis_0.Enable := gMpDelta4AxisEnable;
		MpDelta4Axis_0.Jog := gMpDelta4AxisJog;

	END_IF
END_ACTION
```

#### AxisConfig.st
```iecst
ACTION AxisConfigAction:
	MpDelta4Axis_0.MpLink     := ADR(g4AxDeltaA);
	MpDelta4Axis_0.Parameters := ADR(DeltaParameters);
	MpDelta4Axis_0();

	MpAxisBasic_0.MpLink     := ADR(gAxis_1);
	MpAxisBasic_0.Parameters := ADR(AxisParameters_0);
	MpAxisBasic_0();

	MpAxisBasic_1.MpLink     := ADR(gAxis_2);
	MpAxisBasic_1.Parameters := ADR(AxisParameters_1);
	MpAxisBasic_1();

	MpAxisBasic_Q1.MpLink := ADR(gAxisQ1);
	MpAxisBasic_Q1.Parameters := ADR(homingModeQ1);
	MpAxisBasic_Q1();

	MpAxisBasic_Q2.MpLink := ADR(gAxisQ2);
	MpAxisBasic_Q2.Parameters := ADR(homingModeQ2);
	MpAxisBasic_Q2();

	MpAxisBasic_Q3.MpLink := ADR(gAxisQ3);
	MpAxisBasic_Q3.Parameters := ADR(homingModeQ3);
	MpAxisBasic_Q3();

	MpAxisBasic_Q4.MpLink := ADR(gAxisQ4);
	MpAxisBasic_Q4.Parameters := ADR(homingModeQ4);
	MpAxisBasic_Q4();
END_ACTION
```
